;ENDFOLD
;FOLD LIN P197 CONT Vel=0.055 m/s CPDATP197 Tool[2] Base[8] ;%{PE}
;FOLD Parameters ;%{h}
;Params IlfProvider=kukaroboter.basistech.inlineforms.movement.old; Kuka.IsGlobalPoint=False; Kuka.PointName=P197; Kuka.BlendingEnabled=TRUE; Kuka.MoveDataName=CPDATP197; Kuka.VelocityPath=0.055; Kuka.CurrentCDSetIndex=0; Kuka.MovementParameterFieldEnabled=True; IlfCommand=LIN
;ENDFOLD
$BWDSTART = FALSE
LDAT_ACT=LCPDATP197
FDAT_ACT=FP197
BAS (#CP_PARAMS,0.055)
SET_CD_PARAMS (0)
LIN XP197 C_DIS

;ENDFOLD
;FOLD LIN P198 CONT Vel=0.12 m/s CPDATP198 Tool[2] Base[8] ;%{PE}
;FOLD Parameters ;%{h}
;Params IlfProvider=kukaroboter.basistech.inlineforms.movement.old; Kuka.IsGlobalPoint=False; Kuka.PointName=P198; Kuka.BlendingEnabled=TRUE; Kuka.MoveDataName=CPDATP198; Kuka.VelocityPath=0.12; Kuka.CurrentCDSetIndex=0; Kuka.MovementParameterFieldEnabled=True; IlfCommand=LIN
;ENDFOLD
$BWDSTART = FALSE
LDAT_ACT=LCPDATP198
FDAT_ACT=FP198
BAS (#CP_PARAMS,0.12)
SET_CD_PARAMS (0)
LIN XP198 C_DIS

;ENDFOLD
;FOLD LIN P199 CONT Vel=0.12 m/s CPDATP199 Tool[2] Base[8] ;%{PE}
;FOLD Parameters ;%{h}
;Params IlfProvider=kukaroboter.basistech.inlineforms.movement.old; Kuka.IsGlobalPoint=False; Kuka.PointName=P199; Kuka.BlendingEnabled=TRUE; Kuka.MoveDataName=CPDATP199; Kuka.VelocityPath=0.12; Kuka.CurrentCDSetIndex=0; Kuka.MovementParameterFieldEnabled=True; IlfCommand=LIN
;ENDFOLD
$BWDSTART = FALSE
LDAT_ACT=LCPDATP199
FDAT_ACT=FP199
BAS (#CP_PARAMS,0.12)
SET_CD_PARAMS (0)
LIN XP199 C_DIS

;ENDFOLD
;FOLD LIN P200 CONT Vel=0.12 m/s CPDATP200 Tool[2] Base[8] ;%{PE}
;FOLD Parameters ;%{h}
;Params IlfProvider=kukaroboter.basistech.inlineforms.movement.old; Kuka.IsGlobalPoint=False; Kuka.PointName=P200; Kuka.BlendingEnabled=TRUE; Kuka.MoveDataName=CPDATP200; Kuka.VelocityPath=0.12; Kuka.CurrentCDSetIndex=0; Kuka.MovementParameterFieldEnabled=True; IlfCommand=LIN
;ENDFOLD
$BWDSTART = FALSE
LDAT_ACT=LCPDATP200
FDAT_ACT=FP200
BAS (#CP_PARAMS,0.12)
SET_CD_PARAMS (0)
LIN XP200 C_DIS

;ENDFOLD
;FOLD LIN P201 CONT Vel=0.12 m/s CPDATP201 Tool[2] Base[8] ;%{PE}
;FOLD Parameters ;%{h}
;Params IlfProvider=kukaroboter.basistech.inlineforms.movement.old; Kuka.IsGlobalPoint=False; Kuka.PointName=P201; Kuka.BlendingEnabled=TRUE; Kuka.MoveDataName=CPDATP201; Kuka.VelocityPath=0.12; Kuka.CurrentCDSetIndex=0; Kuka.MovementParameterFieldEnabled=True; IlfCommand=LIN
;ENDFOLD
$BWDSTART = FALSE
LDAT_ACT=LCPDATP201
FDAT_ACT=FP201
BAS (#CP_PARAMS,0.12)
SET_CD_PARAMS (0)
LIN XP201 C_DIS

;ENDFOLD
;FOLD LIN P202 CONT Vel=0.081 m/s CPDATP202 Tool[2] Base[8] ;%{PE}
;FOLD Parameters ;%{h}
;Params IlfProvider=kukaroboter.basistech.inlineforms.movement.old; Kuka.IsGlobalPoint=False; Kuka.PointName=P202; Kuka.BlendingEnabled=TRUE; Kuka.MoveDataName=CPDATP202; Kuka.VelocityPath=0.081; Kuka.CurrentCDSetIndex=0; Kuka.MovementParameterFieldEnabled=True; IlfCommand=LIN
;ENDFOLD
$BWDSTART = FALSE
LDAT_ACT=LCPDATP202
FDAT_ACT=FP202
BAS (#CP_PARAMS,0.081)
SET_CD_PARAMS (0)
LIN XP202 C_DIS

;ENDFOLD
;FOLD LIN P203 CONT Vel=0.081 m/s CPDATP203 Tool[2] Base[8] ;%{PE}
;FOLD Parameters ;%{h}
;Params IlfProvider=kukaroboter.basistech.inlineforms.movement.old; Kuka.IsGlobalPoint=False; Kuka.PointName=P203; Kuka.BlendingEnabled=TRUE; Kuka.MoveDataName=CPDATP203; Kuka.VelocityPath=0.081; Kuka.CurrentCDSetIndex=0; Kuka.MovementParameterFieldEnabled=True; IlfCommand=LIN
;ENDFOLD
$BWDSTART = FALSE
LDAT_ACT=LCPDATP203
FDAT_ACT=FP203
BAS (#CP_PARAMS,0.081)
SET_CD_PARAMS (0)
LIN XP203 C_DIS

;ENDFOLD
;FOLD LIN P204 CONT Vel=0.081 m/s CPDATP204 Tool[2] Base[8] ;%{PE}
;FOLD Parameters ;%{h}
;Params IlfProvider=kukaroboter.basistech.inlineforms.movement.old; Kuka.IsGlobalPoint=False; Kuka.PointName=P204; Kuka.BlendingEnabled=TRUE; Kuka.MoveDataName=CPDATP204; Kuka.VelocityPath=0.081; Kuka.CurrentCDSetIndex=0; Kuka.MovementParameterFieldEnabled=True; IlfCommand=LIN
;ENDFOLD
$BWDSTART = FALSE
LDAT_ACT=LCPDATP204
FDAT_ACT=FP204
BAS (#CP_PARAMS,0.081)
SET_CD_PARAMS (0)
LIN XP204 C_DIS

;ENDFOLD
;FOLD LIN P205 CONT Vel=0.081 m/s CPDATP205 Tool[2] Base[8] ;%{PE}
;FOLD Parameters ;%{h}
;Params IlfProvider=kukaroboter.basistech.inlineforms.movement.old; Kuka.IsGlobalPoint=False; Kuka.PointName=P205; Kuka.BlendingEnabled=TRUE; Kuka.MoveDataName=CPDATP205; Kuka.VelocityPath=0.081; Kuka.CurrentCDSetIndex=0; Kuka.MovementParameterFieldEnabled=True; IlfCommand=LIN
;ENDFOLD
$BWDSTART = FALSE
LDAT_ACT=LCPDATP205
FDAT_ACT=FP205
BAS (#CP_PARAMS,0.081)
SET_CD_PARAMS (0)
LIN XP205 C_DIS

;ENDFOLD
;FOLD LIN P206 CONT Vel=0.147 m/s CPDATP206 Tool[2] Base[8] ;%{PE}
;FOLD Parameters ;%{h}
;Params IlfProvider=kukaroboter.basistech.inlineforms.movement.old; Kuka.IsGlobalPoint=False; Kuka.PointName=P206; Kuka.BlendingEnabled=TRUE; Kuka.MoveDataName=CPDATP206; Kuka.VelocityPath=0.147; Kuka.CurrentCDSetIndex=0; Kuka.MovementParameterFieldEnabled=True; IlfCommand=LIN
;ENDFOLD
$BWDSTART = FALSE
LDAT_ACT=LCPDATP206
FDAT_ACT=FP206
BAS (#CP_PARAMS,0.147)
SET_CD_PARAMS (0)
LIN XP206 C_DIS

;ENDFOLD
;FOLD LIN P207 CONT Vel=0.147 m/s CPDATP207 Tool[2] Base[8] ;%{PE}
;FOLD Parameters ;%{h}
;Params IlfProvider=kukaroboter.basistech.inlineforms.movement.old; Kuka.IsGlobalPoint=False; Kuka.PointName=P207; Kuka.BlendingEnabled=TRUE; Kuka.MoveDataName=CPDATP207; Kuka.VelocityPath=0.147; Kuka.CurrentCDSetIndex=0; Kuka.MovementParameterFieldEnabled=True; IlfCommand=LIN
;ENDFOLD
$BWDSTART = FALSE
LDAT_ACT=LCPDATP207
FDAT_ACT=FP207
BAS (#CP_PARAMS,0.147)
SET_CD_PARAMS (0)
LIN XP207 C_DIS

;ENDFOLD
;FOLD LIN P208 CONT Vel=0.147 m/s CPDATP208 Tool[2] Base[8] ;%{PE}
;FOLD Parameters ;%{h}
;Params IlfProvider=kukaroboter.basistech.inlineforms.movement.old; Kuka.IsGlobalPoint=False; Kuka.PointName=P208; Kuka.BlendingEnabled=TRUE; Kuka.MoveDataName=CPDATP208; Kuka.VelocityPath=0.147; Kuka.CurrentCDSetIndex=0; Kuka.MovementParameterFieldEnabled=True; IlfCommand=LIN
;ENDFOLD
$BWDSTART = FALSE
LDAT_ACT=LCPDATP208
FDAT_ACT=FP208
BAS (#CP_PARAMS,0.147)
SET_CD_PARAMS (0)
LIN XP208 C_DIS

;ENDFOLD
;FOLD LIN P209 CONT Vel=0.147 m/s CPDATP209 Tool[2] Base[8] ;%{PE}
;FOLD Parameters ;%{h}
;Params IlfProvider=kukaroboter.basistech.inlineforms.movement.old; Kuka.IsGlobalPoint=False; Kuka.PointName=P209; Kuka.BlendingEnabled=TRUE; Kuka.MoveDataName=CPDATP209; Kuka.VelocityPath=0.147; Kuka.CurrentCDSetIndex=0; Kuka.MovementParameterFieldEnabled=True; IlfCommand=LIN
;ENDFOLD
$BWDSTART = FALSE
LDAT_ACT=LCPDATP209
FDAT_ACT=FP209
BAS (#CP_PARAMS,0.147)
SET_CD_PARAMS (0)
LIN XP209 C_DIS

;ENDFOLD
;FOLD LIN P210 CONT Vel=0.076 m/s CPDATP210 Tool[2] Base[8] ;%{PE}
;FOLD Parameters ;%{h}
;Params IlfProvider=kukaroboter.basistech.inlineforms.movement.old; Kuka.IsGlobalPoint=False; Kuka.PointName=P210; Kuka.BlendingEnabled=TRUE; Kuka.MoveDataName=CPDATP210; Kuka.VelocityPath=0.076; Kuka.CurrentCDSetIndex=0; Kuka.MovementParameterFieldEnabled=True; IlfCommand=LIN
;ENDFOLD
$BWDSTART = FALSE
LDAT_ACT=LCPDATP210
FDAT_ACT=FP210
BAS (#CP_PARAMS,0.076)
SET_CD_PARAMS (0)
LIN XP210 C_DIS

;ENDFOLD
;FOLD LIN P211 CONT Vel=0.076 m/s CPDATP211 Tool[2] Base[8] ;%{PE}
;FOLD Parameters ;%{h}
;Params IlfProvider=kukaroboter.basistech.inlineforms.movement.old; Kuka.IsGlobalPoint=False; Kuka.PointName=P211; Kuka.BlendingEnabled=TRUE; Kuka.MoveDataName=CPDATP211; Kuka.VelocityPath=0.076; Kuka.CurrentCDSetIndex=0; Kuka.MovementParameterFieldEnabled=True; IlfCommand=LIN
;ENDFOLD
$BWDSTART = FALSE
LDAT_ACT=LCPDATP211
FDAT_ACT=FP211
BAS (#CP_PARAMS,0.076)
SET_CD_PARAMS (0)
LIN XP211 C_DIS

;ENDFOLD
;FOLD LIN P212 CONT Vel=0.076 m/s CPDATP212 Tool[2] Base[8] ;%{PE}
;FOLD Parameters ;%{h}
;Params IlfProvider=kukaroboter.basistech.inlineforms.movement.old; Kuka.IsGlobalPoint=False; Kuka.PointName=P212; Kuka.BlendingEnabled=TRUE; Kuka.MoveDataName=CPDATP212; Kuka.VelocityPath=0.076; Kuka.CurrentCDSetIndex=0; Kuka.MovementParameterFieldEnabled=True; IlfCommand=LIN
;ENDFOLD
$BWDSTART = FALSE
LDAT_ACT=LCPDATP212
FDAT_ACT=FP212
BAS (#CP_PARAMS,0.076)
SET_CD_PARAMS (0)
LIN XP212 C_DIS

;ENDFOLD
;FOLD LIN P213 CONT Vel=0.076 m/s CPDATP213 Tool[2] Base[8] ;%{PE}
;FOLD Parameters ;%{h}
;Params IlfProvider=kukaroboter.basistech.inlineforms.movement.old; Kuka.IsGlobalPoint=False; Kuka.PointName=P213; Kuka.BlendingEnabled=TRUE; Kuka.MoveDataName=CPDATP213; Kuka.VelocityPath=0.076; Kuka.CurrentCDSetIndex=0; Kuka.MovementParameterFieldEnabled=True; IlfCommand=LIN
;ENDFOLD
$BWDSTART = FALSE
LDAT_ACT=LCPDATP213
FDAT_ACT=FP213
BAS (#CP_PARAMS,0.076)
SET_CD_PARAMS (0)
LIN XP213 C_DIS

;ENDFOLD
;FOLD LIN P214 CONT Vel=0.126 m/s CPDATP214 Tool[2] Base[8] ;%{PE}
;FOLD Parameters ;%{h}
;Params IlfProvider=kukaroboter.basistech.inlineforms.movement.old; Kuka.IsGlobalPoint=False; Kuka.PointName=P214; Kuka.BlendingEnabled=TRUE; Kuka.MoveDataName=CPDATP214; Kuka.VelocityPath=0.126; Kuka.CurrentCDSetIndex=0; Kuka.MovementParameterFieldEnabled=True; IlfCommand=LIN
;ENDFOLD
$BWDSTART = FALSE
LDAT_ACT=LCPDATP214
FDAT_ACT=FP214
BAS (#CP_PARAMS,0.126)
SET_CD_PARAMS (0)
LIN XP214 C_DIS

;ENDFOLD
;FOLD LIN P215 CONT Vel=0.126 m/s CPDATP215 Tool[2] Base[8] ;%{PE}
;FOLD Parameters ;%{h}
;Params IlfProvider=kukaroboter.basistech.inlineforms.movement.old; Kuka.IsGlobalPoint=False; Kuka.PointName=P215; Kuka.BlendingEnabled=TRUE; Kuka.MoveDataName=CPDATP215; Kuka.VelocityPath=0.126; Kuka.CurrentCDSetIndex=0; Kuka.MovementParameterFieldEnabled=True; IlfCommand=LIN
;ENDFOLD
$BWDSTART = FALSE
LDAT_ACT=LCPDATP215
FDAT_ACT=FP215
BAS (#CP_PARAMS,0.126)
SET_CD_PARAMS (0)
LIN XP215 C_DIS

;ENDFOLD
;FOLD LIN P216 CONT Vel=0.126 m/s CPDATP216 Tool[2] Base[8] ;%{PE}
;FOLD Parameters ;%{h}
;Params IlfProvider=kukaroboter.basistech.inlineforms.movement.old; Kuka.IsGlobalPoint=False; Kuka.PointName=P216; Kuka.BlendingEnabled=TRUE; Kuka.MoveDataName=CPDATP216; Kuka.VelocityPath=0.126; Kuka.CurrentCDSetIndex=0; Kuka.MovementParameterFieldEnabled=True; IlfCommand=LIN
;ENDFOLD
$BWDSTART = FALSE
LDAT_ACT=LCPDATP216
FDAT_ACT=FP216
BAS (#CP_PARAMS,0.126)
SET_CD_PARAMS (0)
LIN XP216 C_DIS

;ENDFOLD
;FOLD LIN P217 CONT Vel=0.126 m/s CPDATP217 Tool[2] Base[8] ;%{PE}
;FOLD Parameters ;%{h}
;Params IlfProvider=kukaroboter.basistech.inlineforms.movement.old; Kuka.IsGlobalPoint=False; Kuka.PointName=P217; Kuka.BlendingEnabled=TRUE; Kuka.MoveDataName=CPDATP217; Kuka.VelocityPath=0.126; Kuka.CurrentCDSetIndex=0; Kuka.MovementParameterFieldEnabled=True; IlfCommand=LIN
;ENDFOLD
$BWDSTART = FALSE
LDAT_ACT=LCPDATP217
FDAT_ACT=FP217
BAS (#CP_PARAMS,0.126)
SET_CD_PARAMS (0)
LIN XP217 C_DIS

;ENDFOLD
;FOLD LIN P218 CONT Vel=0.13 m/s CPDATP218 Tool[2] Base[8] ;%{PE}
;FOLD Parameters ;%{h}
;Params IlfProvider=kukaroboter.basistech.inlineforms.movement.old; Kuka.IsGlobalPoint=False; Kuka.PointName=P218; Kuka.BlendingEnabled=TRUE; Kuka.MoveDataName=CPDATP218; Kuka.VelocityPath=0.13; Kuka.CurrentCDSetIndex=0; Kuka.MovementParameterFieldEnabled=True; IlfCommand=LIN
;ENDFOLD
$BWDSTART = FALSE
LDAT_ACT=LCPDATP218
FDAT_ACT=FP218
BAS (#CP_PARAMS,0.13)
SET_CD_PARAMS (0)
LIN XP218 C_DIS

;ENDFOLD
;FOLD LIN P219 CONT Vel=0.13 m/s CPDATP219 Tool[2] Base[8] ;%{PE}
;FOLD Parameters ;%{h}
;Params IlfProvider=kukaroboter.basistech.inlineforms.movement.old; Kuka.IsGlobalPoint=False; Kuka.PointName=P219; Kuka.BlendingEnabled=TRUE; Kuka.MoveDataName=CPDATP219; Kuka.VelocityPath=0.13; Kuka.CurrentCDSetIndex=0; Kuka.MovementParameterFieldEnabled=True; IlfCommand=LIN
;ENDFOLD
$BWDSTART = FALSE
LDAT_ACT=LCPDATP219
FDAT_ACT=FP219
BAS (#CP_PARAMS,0.13)
SET_CD_PARAMS (0)
LIN XP219 C_DIS

;ENDFOLD
;FOLD LIN P220 CONT Vel=0.13 m/s CPDATP220 Tool[2] Base[8] ;%{PE}
;FOLD Parameters ;%{h}
;Params IlfProvider=kukaroboter.basistech.inlineforms.movement.old; Kuka.IsGlobalPoint=False; Kuka.PointName=P220; Kuka.BlendingEnabled=TRUE; Kuka.MoveDataName=CPDATP220; Kuka.VelocityPath=0.13; Kuka.CurrentCDSetIndex=0; Kuka.MovementParameterFieldEnabled=True; IlfCommand=LIN
;ENDFOLD
$BWDSTART = FALSE
LDAT_ACT=LCPDATP220
FDAT_ACT=FP220
BAS (#CP_PARAMS,0.13)
SET_CD_PARAMS (0)
LIN XP220 C_DIS

;ENDFOLD
;FOLD LIN P221 CONT Vel=0.13 m/s CPDATP221 Tool[2] Base[8] ;%{PE}
;FOLD Parameters ;%{h}
;Params IlfProvider=kukaroboter.basistech.inlineforms.movement.old; Kuka.IsGlobalPoint=False; Kuka.PointName=P221; Kuka.BlendingEnabled=TRUE; Kuka.MoveDataName=CPDATP221; Kuka.VelocityPath=0.13; Kuka.CurrentCDSetIndex=0; Kuka.MovementParameterFieldEnabled=True; IlfCommand=LIN
;ENDFOLD
$BWDSTART = FALSE
LDAT_ACT=LCPDATP221
FDAT_ACT=FP221
BAS (#CP_PARAMS,0.13)
SET_CD_PARAMS (0)
LIN XP221 C_DIS

;ENDFOLD
;FOLD LIN P222 CONT Vel=0.106 m/s CPDATP222 Tool[2] Base[8] ;%{PE}
;FOLD Parameters ;%{h}
;Params IlfProvider=kukaroboter.basistech.inlineforms.movement.old; Kuka.IsGlobalPoint=False; Kuka.PointName=P222; Kuka.BlendingEnabled=TRUE; Kuka.MoveDataName=CPDATP222; Kuka.VelocityPath=0.106; Kuka.CurrentCDSetIndex=0; Kuka.MovementParameterFieldEnabled=True; IlfCommand=LIN
;ENDFOLD
$BWDSTART = FALSE
LDAT_ACT=LCPDATP222
FDAT_ACT=FP222
BAS (#CP_PARAMS,0.106)
SET_CD_PARAMS (0)
LIN XP222 C_DIS

;ENDFOLD
;FOLD LIN P223 CONT Vel=0.106 m/s CPDATP223 Tool[2] Base[8] ;%{PE}
;FOLD Parameters ;%{h}
;Params IlfProvider=kukaroboter.basistech.inlineforms.movement.old; Kuka.IsGlobalPoint=False; Kuka.PointName=P223; Kuka.BlendingEnabled=TRUE; Kuka.MoveDataName=CPDATP223; Kuka.VelocityPath=0.106; Kuka.CurrentCDSetIndex=0; Kuka.MovementParameterFieldEnabled=True; IlfCommand=LIN
;ENDFOLD
$BWDSTART = FALSE
LDAT_ACT=LCPDATP223
FDAT_ACT=FP223
BAS (#CP_PARAMS,0.106)
SET_CD_PARAMS (0)
LIN XP223 C_DIS

;ENDFOLD
;FOLD LIN P224 CONT Vel=0.106 m/s CPDATP224 Tool[2] Base[8] ;%{PE}
;FOLD Parameters ;%{h}
;Params IlfProvider=kukaroboter.basistech.inlineforms.movement.old; Kuka.IsGlobalPoint=False; Kuka.PointName=P224; Kuka.BlendingEnabled=TRUE; Kuka.MoveDataName=CPDATP224; Kuka.VelocityPath=0.106; Kuka.CurrentCDSetIndex=0; Kuka.MovementParameterFieldEnabled=True; IlfCommand=LIN
;ENDFOLD
$BWDSTART = FALSE
LDAT_ACT=LCPDATP224
FDAT_ACT=FP224
BAS (#CP_PARAMS,0.106)
SET_CD_PARAMS (0)
LIN XP224 C_DIS

;ENDFOLD
;FOLD LIN P225 CONT Vel=0.106 m/s CPDATP225 Tool[2] Base[8] ;%{PE}
;FOLD Parameters ;%{h}
;Params IlfProvider=kukaroboter.basistech.inlineforms.movement.old; Kuka.IsGlobalPoint=False; Kuka.PointName=P225; Kuka.BlendingEnabled=TRUE; Kuka.MoveDataName=CPDATP225; Kuka.VelocityPath=0.106; Kuka.CurrentCDSetIndex=0; Kuka.MovementParameterFieldEnabled=True; IlfCommand=LIN
;ENDFOLD
$BWDSTART = FALSE
LDAT_ACT=LCPDATP225
FDAT_ACT=FP225
BAS (#CP_PARAMS,0.106)
SET_CD_PARAMS (0)
LIN XP225 C_DIS

;ENDFOLD
;FOLD LIN P226 CONT Vel=0.145 m/s CPDATP226 Tool[2] Base[8] ;%{PE}
;FOLD Parameters ;%{h}
;Params IlfProvider=kukaroboter.basistech.inlineforms.movement.old; Kuka.IsGlobalPoint=False; Kuka.PointName=P226; Kuka.BlendingEnabled=TRUE; Kuka.MoveDataName=CPDATP226; Kuka.VelocityPath=0.145; Kuka.CurrentCDSetIndex=0; Kuka.MovementParameterFieldEnabled=True; IlfCommand=LIN
;ENDFOLD
$BWDSTART = FALSE
LDAT_ACT=LCPDATP226
FDAT_ACT=FP226
BAS (#CP_PARAMS,0.145)
SET_CD_PARAMS (0)
LIN XP226 C_DIS

;ENDFOLD
;FOLD LIN P227 CONT Vel=0.145 m/s CPDATP227 Tool[2] Base[8] ;%{PE}
;FOLD Parameters ;%{h}
;Params IlfProvider=kukaroboter.basistech.inlineforms.movement.old; Kuka.IsGlobalPoint=False; Kuka.PointName=P227; Kuka.BlendingEnabled=TRUE; Kuka.MoveDataName=CPDATP227; Kuka.VelocityPath=0.145; Kuka.CurrentCDSetIndex=0; Kuka.MovementParameterFieldEnabled=True; IlfCommand=LIN
;ENDFOLD
$BWDSTART = FALSE
LDAT_ACT=LCPDATP227
FDAT_ACT=FP227
BAS (#CP_PARAMS,0.145)
SET_CD_PARAMS (0)
LIN XP227 C_DIS

;ENDFOLD
;FOLD LIN P228 CONT Vel=0.145 m/s CPDATP228 Tool[2] Base[8] ;%{PE}
;FOLD Parameters ;%{h}
;Params IlfProvider=kukaroboter.basistech.inlineforms.movement.old; Kuka.IsGlobalPoint=False; Kuka.PointName=P228; Kuka.BlendingEnabled=TRUE; Kuka.MoveDataName=CPDATP228; Kuka.VelocityPath=0.145; Kuka.CurrentCDSetIndex=0; Kuka.MovementParameterFieldEnabled=True; IlfCommand=LIN
;ENDFOLD
$BWDSTART = FALSE
LDAT_ACT=LCPDATP228
FDAT_ACT=FP228
BAS (#CP_PARAMS,0.145)
SET_CD_PARAMS (0)
LIN XP228 C_DIS

;ENDFOLD
;FOLD LIN P229 CONT Vel=0.145 m/s CPDATP229 Tool[2] Base[8] ;%{PE}
;FOLD Parameters ;%{h}
;Params IlfProvider=kukaroboter.basistech.inlineforms.movement.old; Kuka.IsGlobalPoint=False; Kuka.PointName=P229; Kuka.BlendingEnabled=TRUE; Kuka.MoveDataName=CPDATP229; Kuka.VelocityPath=0.145; Kuka.CurrentCDSetIndex=0; Kuka.MovementParameterFieldEnabled=True; IlfCommand=LIN
;ENDFOLD
$BWDSTART = FALSE
LDAT_ACT=LCPDATP229
FDAT_ACT=FP229
BAS (#CP_PARAMS,0.145)
SET_CD_PARAMS (0)
LIN XP229 C_DIS

;ENDFOLD
;FOLD LIN P230 CONT Vel=0.1 m/s CPDATP230 Tool[2] Base[8] ;%{PE}
;FOLD Parameters ;%{h}
;Params IlfProvider=kukaroboter.basistech.inlineforms.movement.old; Kuka.IsGlobalPoint=False; Kuka.PointName=P230; Kuka.BlendingEnabled=TRUE; Kuka.MoveDataName=CPDATP230; Kuka.VelocityPath=0.1; Kuka.CurrentCDSetIndex=0; Kuka.MovementParameterFieldEnabled=True; IlfCommand=LIN
;ENDFOLD
$BWDSTART = FALSE
LDAT_ACT=LCPDATP230
FDAT_ACT=FP230
BAS (#CP_PARAMS,0.1)
SET_CD_PARAMS (0)
LIN XP230 C_DIS

;ENDFOLD
;FOLD LIN P231 CONT Vel=0.1 m/s CPDATP231 Tool[2] Base[8] ;%{PE}
;FOLD Parameters ;%{h}
;Params IlfProvider=kukaroboter.basistech.inlineforms.movement.old; Kuka.IsGlobalPoint=False; Kuka.PointName=P231; Kuka.BlendingEnabled=TRUE; Kuka.MoveDataName=CPDATP231; Kuka.VelocityPath=0.1; Kuka.CurrentCDSetIndex=0; Kuka.MovementParameterFieldEnabled=True; IlfCommand=LIN
;ENDFOLD
$BWDSTART = FALSE
LDAT_ACT=LCPDATP231
FDAT_ACT=FP231
BAS (#CP_PARAMS,0.1)
SET_CD_PARAMS (0)
LIN XP231 C_DIS

;ENDFOLD
;FOLD LIN P232 CONT Vel=0.1 m/s CPDATP232 Tool[2] Base[8] ;%{PE}
;FOLD Parameters ;%{h}
;Params IlfProvider=kukaroboter.basistech.inlineforms.movement.old; Kuka.IsGlobalPoint=False; Kuka.PointName=P232; Kuka.BlendingEnabled=TRUE; Kuka.MoveDataName=CPDATP232; Kuka.VelocityPath=0.1; Kuka.CurrentCDSetIndex=0; Kuka.MovementParameterFieldEnabled=True; IlfCommand=LIN
;ENDFOLD
$BWDSTART = FALSE
LDAT_ACT=LCPDATP232
FDAT_ACT=FP232
BAS (#CP_PARAMS,0.1)
SET_CD_PARAMS (0)
LIN XP232 C_DIS

;ENDFOLD
;FOLD LIN P233 CONT Vel=0.1 m/s CPDATP233 Tool[2] Base[8] ;%{PE}
;FOLD Parameters ;%{h}
;Params IlfProvider=kukaroboter.basistech.inlineforms.movement.old; Kuka.IsGlobalPoint=False; Kuka.PointName=P233; Kuka.BlendingEnabled=TRUE; Kuka.MoveDataName=CPDATP233; Kuka.VelocityPath=0.1; Kuka.CurrentCDSetIndex=0; Kuka.MovementParameterFieldEnabled=True; IlfCommand=LIN
;ENDFOLD
$BWDSTART = FALSE
LDAT_ACT=LCPDATP233
FDAT_ACT=FP233
BAS (#CP_PARAMS,0.1)
SET_CD_PARAMS (0)
LIN XP233 C_DIS

;ENDFOLD
;FOLD LIN P234 CONT Vel=0.13 m/s CPDATP234 Tool[2] Base[8] ;%{PE}
;FOLD Parameters ;%{h}
;Params IlfProvider=kukaroboter.basistech.inlineforms.movement.old; Kuka.IsGlobalPoint=False; Kuka.PointName=P234; Kuka.BlendingEnabled=TRUE; Kuka.MoveDataName=CPDATP234; Kuka.VelocityPath=0.13; Kuka.CurrentCDSetIndex=0; Kuka.MovementParameterFieldEnabled=True; IlfCommand=LIN
;ENDFOLD
$BWDSTART = FALSE
LDAT_ACT=LCPDATP234
FDAT_ACT=FP234
BAS (#CP_PARAMS,0.13)
SET_CD_PARAMS (0)
LIN XP234 C_DIS

;ENDFOLD
;FOLD LIN P235 CONT Vel=0.13 m/s CPDATP235 Tool[2] Base[8] ;%{PE}
;FOLD Parameters ;%{h}
;Params IlfProvider=kukaroboter.basistech.inlineforms.movement.old; Kuka.IsGlobalPoint=False; Kuka.PointName=P235; Kuka.BlendingEnabled=TRUE; Kuka.MoveDataName=CPDATP235; Kuka.VelocityPath=0.13; Kuka.CurrentCDSetIndex=0; Kuka.MovementParameterFieldEnabled=True; IlfCommand=LIN
;ENDFOLD
$BWDSTART = FALSE
LDAT_ACT=LCPDATP235
FDAT_ACT=FP235
BAS (#CP_PARAMS,0.13)
SET_CD_PARAMS (0)
LIN XP235 C_DIS

;ENDFOLD
;FOLD LIN P236 CONT Vel=0.13 m/s CPDATP236 Tool[2] Base[8] ;%{PE}
;FOLD Parameters ;%{h}
;Params IlfProvider=kukaroboter.basistech.inlineforms.movement.old; Kuka.IsGlobalPoint=False; Kuka.PointName=P236; Kuka.BlendingEnabled=TRUE; Kuka.MoveDataName=CPDATP236; Kuka.VelocityPath=0.13; Kuka.CurrentCDSetIndex=0; Kuka.MovementParameterFieldEnabled=True; IlfCommand=LIN
;ENDFOLD
$BWDSTART = FALSE
LDAT_ACT=LCPDATP236
FDAT_ACT=FP236
BAS (#CP_PARAMS,0.13)
SET_CD_PARAMS (0)
LIN XP236 C_DIS

;ENDFOLD
;FOLD LIN P237 CONT Vel=0.13 m/s CPDATP237 Tool[2] Base[8] ;%{PE}
;FOLD Parameters ;%{h}
;Params IlfProvider=kukaroboter.basistech.inlineforms.movement.old; Kuka.IsGlobalPoint=False; Kuka.PointName=P237; Kuka.BlendingEnabled=TRUE; Kuka.MoveDataName=CPDATP237; Kuka.VelocityPath=0.13; Kuka.CurrentCDSetIndex=0; Kuka.MovementParameterFieldEnabled=True; IlfCommand=LIN
;ENDFOLD
$BWDSTART = FALSE
LDAT_ACT=LCPDATP237
FDAT_ACT=FP237
BAS (#CP_PARAMS,0.13)
SET_CD_PARAMS (0)
LIN XP237 C_DIS

;ENDFOLD
;FOLD LIN P238 CONT Vel=0.091 m/s CPDATP238 Tool[2] Base[8] ;%{PE}
;FOLD Parameters ;%{h}
;Params IlfProvider=kukaroboter.basistech.inlineforms.movement.old; Kuka.IsGlobalPoint=False; Kuka.PointName=P238; Kuka.BlendingEnabled=TRUE; Kuka.MoveDataName=CPDATP238; Kuka.VelocityPath=0.091; Kuka.CurrentCDSetIndex=0; Kuka.MovementParameterFieldEnabled=True; IlfCommand=LIN
;ENDFOLD
$BWDSTART = FALSE
LDAT_ACT=LCPDATP238
FDAT_ACT=FP238
BAS (#CP_PARAMS,0.091)
SET_CD_PARAMS (0)
LIN XP238 C_DIS

;ENDFOLD
;FOLD LIN P239 CONT Vel=0.091 m/s CPDATP239 Tool[2] Base[8] ;%{PE}
;FOLD Parameters ;%{h}
;Params IlfProvider=kukaroboter.basistech.inlineforms.movement.old; Kuka.IsGlobalPoint=False; Kuka.PointName=P239; Kuka.BlendingEnabled=TRUE; Kuka.MoveDataName=CPDATP239; Kuka.VelocityPath=0.091; Kuka.CurrentCDSetIndex=0; Kuka.MovementParameterFieldEnabled=True; IlfCommand=LIN
;ENDFOLD
$BWDSTART = FALSE
LDAT_ACT=LCPDATP239
FDAT_ACT=FP239
BAS (#CP_PARAMS,0.091)
SET_CD_PARAMS (0)
LIN XP239 C_DIS

;ENDFOLD
;FOLD LIN P240 CONT Vel=0.091 m/s CPDATP240 Tool[2] Base[8] ;%{PE}
;FOLD Parameters ;%{h}
;Params IlfProvider=kukaroboter.basistech.inlineforms.movement.old; Kuka.IsGlobalPoint=False; Kuka.PointName=P240; Kuka.BlendingEnabled=TRUE; Kuka.MoveDataName=CPDATP240; Kuka.VelocityPath=0.091; Kuka.CurrentCDSetIndex=0; Kuka.MovementParameterFieldEnabled=True; IlfCommand=LIN
;ENDFOLD
$BWDSTART = FALSE
LDAT_ACT=LCPDATP240
FDAT_ACT=FP240
BAS (#CP_PARAMS,0.091)
SET_CD_PARAMS (0)
LIN XP240 C_DIS

;ENDFOLD
;FOLD LIN P241 CONT Vel=0.091 m/s CPDATP241 Tool[2] Base[8] ;%{PE}
;FOLD Parameters ;%{h}
;Params IlfProvider=kukaroboter.basistech.inlineforms.movement.old; Kuka.IsGlobalPoint=False; Kuka.PointName=P241; Kuka.BlendingEnabled=TRUE; Kuka.MoveDataName=CPDATP241; Kuka.VelocityPath=0.091; Kuka.CurrentCDSetIndex=0; Kuka.MovementParameterFieldEnabled=True; IlfCommand=LIN
;ENDFOLD
$BWDSTART = FALSE
LDAT_ACT=LCPDATP241
FDAT_ACT=FP241
BAS (#CP_PARAMS,0.091)
SET_CD_PARAMS (0)
LIN XP241 C_DIS

;ENDFOLD
;FOLD LIN P242 CONT Vel=0.5 m/s CPDATP242 Tool[2] Base[8] ;%{PE}
;FOLD Parameters ;%{h}
;Params IlfProvider=kukaroboter.basistech.inlineforms.movement.old; Kuka.IsGlobalPoint=False; Kuka.PointName=P242; Kuka.BlendingEnabled=TRUE; Kuka.MoveDataName=CPDATP242; Kuka.VelocityPath=0.5; Kuka.CurrentCDSetIndex=0; Kuka.MovementParameterFieldEnabled=True; IlfCommand=LIN
;ENDFOLD
$BWDSTART = FALSE
LDAT_ACT=LCPDATP242
FDAT_ACT=FP242
BAS (#CP_PARAMS,0.5)
SET_CD_PARAMS (0)
LIN XP242 C_DIS

;ENDFOLD
;FOLD LIN P243 CONT Vel=1.0 m/s CPDATP243 Tool[2] Base[8] ;%{PE}
;FOLD Parameters ;%{h}
;Params IlfProvider=kukaroboter.basistech.inlineforms.movement.old; Kuka.IsGlobalPoint=False; Kuka.PointName=P243; Kuka.BlendingEnabled=TRUE; Kuka.MoveDataName=CPDATP243; Kuka.VelocityPath=1.0; Kuka.CurrentCDSetIndex=0; Kuka.MovementParameterFieldEnabled=True; IlfCommand=LIN
;ENDFOLD
$BWDSTART = FALSE
LDAT_ACT=LCPDATP243
FDAT_ACT=FP243
BAS (#CP_PARAMS,1.0)
SET_CD_PARAMS (0)
LIN XP243 C_DIS

;ENDFOLD
;FOLD LIN P244 CONT Vel=1.0 m/s CPDATP244 Tool[2] Base[8] ;%{PE}
;FOLD Parameters ;%{h}
;Params IlfProvider=kukaroboter.basistech.inlineforms.movement.old; Kuka.IsGlobalPoint=False; Kuka.PointName=P244; Kuka.BlendingEnabled=TRUE; Kuka.MoveDataName=CPDATP244; Kuka.VelocityPath=1.0; Kuka.CurrentCDSetIndex=0; Kuka.MovementParameterFieldEnabled=True; IlfCommand=LIN
;ENDFOLD
$BWDSTART = FALSE
LDAT_ACT=LCPDATP244
FDAT_ACT=FP244
BAS (#CP_PARAMS,1.0)
SET_CD_PARAMS (0)
LIN XP244 C_DIS

;ENDFOLD
END
;End of routine {i}

; --- Routine for substrate 3 ---
DEF Routine_3()
;FOLD LIN P245 CONT Vel=1.0 m/s CPDATP245 Tool[2] Base[7] ;%{PE}
;FOLD Parameters ;%{h}
;Params IlfProvider=kukaroboter.basistech.inlineforms.movement.old; Kuka.IsGlobalPoint=False; Kuka.PointName=P245; Kuka.BlendingEnabled=TRUE; Kuka.MoveDataName=CPDATP245; Kuka.VelocityPath=1.0; Kuka.CurrentCDSetIndex=0; Kuka.MovementParameterFieldEnabled=True; IlfCommand=LIN
;ENDFOLD
$BWDSTART = FALSE
LDAT_ACT=LCPDATP245
FDAT_ACT=FP245
BAS (#CP_PARAMS,1.0)
SET_CD_PARAMS (0)
LIN XP245 C_DIS

;ENDFOLD
;FOLD LIN P246 CONT Vel=0.097 m/s CPDATP246 Tool[2] Base[7] ;%{PE}
;FOLD Parameters ;%{h}
;Params IlfProvider=kukaroboter.basistech.inlineforms.movement.old; Kuka.IsGlobalPoint=False; Kuka.PointName=P246; Kuka.BlendingEnabled=TRUE; Kuka.MoveDataName=CPDATP246; Kuka.VelocityPath=0.097; Kuka.CurrentCDSetIndex=0; Kuka.MovementParameterFieldEnabled=True; IlfCommand=LIN
;ENDFOLD
$BWDSTART = FALSE
LDAT_ACT=LCPDATP246
FDAT_ACT=FP246
BAS (#CP_PARAMS,0.097)
SET_CD_PARAMS (0)
LIN XP246 C_DIS

;ENDFOLD
;FOLD LIN P247 CONT Vel=0.097 m/s CPDATP247 Tool[2] Base[7] ;%{PE}
;FOLD Parameters ;%{h}
;Params IlfProvider=kukaroboter.basistech.inlineforms.movement.old; Kuka.IsGlobalPoint=False; Kuka.PointName=P247; Kuka.BlendingEnabled=TRUE; Kuka.MoveDataName=CPDATP247; Kuka.VelocityPath=0.097; Kuka.CurrentCDSetIndex=0; Kuka.MovementParameterFieldEnabled=True; IlfCommand=LIN
;ENDFOLD
$BWDSTART = FALSE
LDAT_ACT=LCPDATP247
FDAT_ACT=FP247
BAS (#CP_PARAMS,0.097)
SET_CD_PARAMS (0)
LIN XP247 C_DIS

;ENDFOLD
;FOLD LIN P248 CONT Vel=0.097 m/s CPDATP248 Tool[2] Base[7] ;%{PE}
;FOLD Parameters ;%{h}
;Params IlfProvider=kukaroboter.basistech.inlineforms.movement.old; Kuka.IsGlobalPoint=False; Kuka.PointName=P248; Kuka.BlendingEnabled=TRUE; Kuka.MoveDataName=CPDATP248; Kuka.VelocityPath=0.097; Kuka.CurrentCDSetIndex=0; Kuka.MovementParameterFieldEnabled=True; IlfCommand=LIN
;ENDFOLD
$BWDSTART = FALSE
LDAT_ACT=LCPDATP248
FDAT_ACT=FP248
BAS (#CP_PARAMS,0.097)
SET_CD_PARAMS (0)
LIN XP248 C_DIS

;ENDFOLD
;FOLD LIN P249 CONT Vel=0.097 m/s CPDATP249 Tool[2] Base[7] ;%{PE}
;FOLD Parameters ;%{h}
;Params IlfProvider=kukaroboter.basistech.inlineforms.movement.old; Kuka.IsGlobalPoint=False; Kuka.PointName=P249; Kuka.BlendingEnabled=TRUE; Kuka.MoveDataName=CPDATP249; Kuka.VelocityPath=0.097; Kuka.CurrentCDSetIndex=0; Kuka.MovementParameterFieldEnabled=True; IlfCommand=LIN
;ENDFOLD
$BWDSTART = FALSE
LDAT_ACT=LCPDATP249
FDAT_ACT=FP249
BAS (#CP_PARAMS,0.097)
SET_CD_PARAMS (0)
LIN XP249 C_DIS

;ENDFOLD
;FOLD LIN P250 CONT Vel=0.144 m/s CPDATP250 Tool[2] Base[7] ;%{PE}
;FOLD Parameters ;%{h}
;Params IlfProvider=kukaroboter.basistech.inlineforms.movement.old; Kuka.IsGlobalPoint=False; Kuka.PointName=P250; Kuka.BlendingEnabled=TRUE; Kuka.MoveDataName=CPDATP250; Kuka.VelocityPath=0.144; Kuka.CurrentCDSetIndex=0; Kuka.MovementParameterFieldEnabled=True; IlfCommand=LIN
;ENDFOLD
$BWDSTART = FALSE
LDAT_ACT=LCPDATP250
FDAT_ACT=FP250
BAS (#CP_PARAMS,0.144)
SET_CD_PARAMS (0)
LIN XP250 C_DIS

;ENDFOLD
;FOLD LIN P251 CONT Vel=0.144 m/s CPDATP251 Tool[2] Base[7] ;%{PE}
;FOLD Parameters ;%{h}
;Params IlfProvider=kukaroboter.basistech.inlineforms.movement.old; Kuka.IsGlobalPoint=False; Kuka.PointName=P251; Kuka.BlendingEnabled=TRUE; Kuka.MoveDataName=CPDATP251; Kuka.VelocityPath=0.144; Kuka.CurrentCDSetIndex=0; Kuka.MovementParameterFieldEnabled=True; IlfCommand=LIN
;ENDFOLD
$BWDSTART = FALSE
LDAT_ACT=LCPDATP251
FDAT_ACT=FP251
BAS (#CP_PARAMS,0.144)
SET_CD_PARAMS (0)
LIN XP251 C_DIS

;ENDFOLD
;FOLD LIN P252 CONT Vel=0.144 m/s CPDATP252 Tool[2] Base[7] ;%{PE}
;FOLD Parameters ;%{h}
;Params IlfProvider=kukaroboter.basistech.inlineforms.movement.old; Kuka.IsGlobalPoint=False; Kuka.PointName=P252; Kuka.BlendingEnabled=TRUE; Kuka.MoveDataName=CPDATP252; Kuka.VelocityPath=0.144; Kuka.CurrentCDSetIndex=0; Kuka.MovementParameterFieldEnabled=True; IlfCommand=LIN
;ENDFOLD
$BWDSTART = FALSE
LDAT_ACT=LCPDATP252
FDAT_ACT=FP252
BAS (#CP_PARAMS,0.144)
SET_CD_PARAMS (0)
LIN XP252 C_DIS

;ENDFOLD
;FOLD LIN P253 CONT Vel=0.144 m/s CPDATP253 Tool[2] Base[7] ;%{PE}
;FOLD Parameters ;%{h}
;Params IlfProvider=kukaroboter.basistech.inlineforms.movement.old; Kuka.IsGlobalPoint=False; Kuka.PointName=P253; Kuka.BlendingEnabled=TRUE; Kuka.MoveDataName=CPDATP253; Kuka.VelocityPath=0.144; Kuka.CurrentCDSetIndex=0; Kuka.MovementParameterFieldEnabled=True; IlfCommand=LIN
;ENDFOLD
$BWDSTART = FALSE
LDAT_ACT=LCPDATP253
FDAT_ACT=FP253
BAS (#CP_PARAMS,0.144)
SET_CD_PARAMS (0)
LIN XP253 C_DIS

;ENDFOLD
;FOLD LIN P254 CONT Vel=0.084 m/s CPDATP254 Tool[2] Base[7] ;%{PE}
;FOLD Parameters ;%{h}
;Params IlfProvider=kukaroboter.basistech.inlineforms.movement.old; Kuka.IsGlobalPoint=False; Kuka.PointName=P254; Kuka.BlendingEnabled=TRUE; Kuka.MoveDataName=CPDATP254; Kuka.VelocityPath=0.084; Kuka.CurrentCDSetIndex=0; Kuka.MovementParameterFieldEnabled=True; IlfCommand=LIN
;ENDFOLD
$BWDSTART = FALSE
LDAT_ACT=LCPDATP254
FDAT_ACT=FP254
BAS (#CP_PARAMS,0.084)
SET_CD_PARAMS (0)
LIN XP254 C_DIS

;ENDFOLD
;FOLD LIN P255 CONT Vel=0.084 m/s CPDATP255 Tool[2] Base[7] ;%{PE}
;FOLD Parameters ;%{h}
;Params IlfProvider=kukaroboter.basistech.inlineforms.movement.old; Kuka.IsGlobalPoint=False; Kuka.PointName=P255; Kuka.BlendingEnabled=TRUE; Kuka.MoveDataName=CPDATP255; Kuka.VelocityPath=0.084; Kuka.CurrentCDSetIndex=0; Kuka.MovementParameterFieldEnabled=True; IlfCommand=LIN
;ENDFOLD
$BWDSTART = FALSE
LDAT_ACT=LCPDATP255
FDAT_ACT=FP255
BAS (#CP_PARAMS,0.084)
SET_CD_PARAMS (0)
LIN XP255 C_DIS

;ENDFOLD
;FOLD LIN P256 CONT Vel=0.084 m/s CPDATP256 Tool[2] Base[7] ;%{PE}
;FOLD Parameters ;%{h}
;Params IlfProvider=kukaroboter.basistech.inlineforms.movement.old; Kuka.IsGlobalPoint=False; Kuka.PointName=P256; Kuka.BlendingEnabled=TRUE; Kuka.MoveDataName=CPDATP256; Kuka.VelocityPath=0.084; Kuka.CurrentCDSetIndex=0; Kuka.MovementParameterFieldEnabled=True; IlfCommand=LIN
;ENDFOLD
$BWDSTART = FALSE
LDAT_ACT=LCPDATP256
FDAT_ACT=FP256
BAS (#CP_PARAMS,0.084)
SET_CD_PARAMS (0)
LIN XP256 C_DIS

;ENDFOLD
;FOLD LIN P257 CONT Vel=0.084 m/s CPDATP257 Tool[2] Base[7] ;%{PE}
;FOLD Parameters ;%{h}
;Params IlfProvider=kukaroboter.basistech.inlineforms.movement.old; Kuka.IsGlobalPoint=False; Kuka.PointName=P257; Kuka.BlendingEnabled=TRUE; Kuka.MoveDataName=CPDATP257; Kuka.VelocityPath=0.084; Kuka.CurrentCDSetIndex=0; Kuka.MovementParameterFieldEnabled=True; IlfCommand=LIN
;ENDFOLD
$BWDSTART = FALSE
LDAT_ACT=LCPDATP257
FDAT_ACT=FP257
BAS (#CP_PARAMS,0.084)
SET_CD_PARAMS (0)
LIN XP257 C_DIS

;ENDFOLD
;FOLD LIN P258 CONT Vel=0.05 m/s CPDATP258 Tool[2] Base[7] ;%{PE}
;FOLD Parameters ;%{h}
;Params IlfProvider=kukaroboter.basistech.inlineforms.movement.old; Kuka.IsGlobalPoint=False; Kuka.PointName=P258; Kuka.BlendingEnabled=TRUE; Kuka.MoveDataName=CPDATP258; Kuka.VelocityPath=0.05; Kuka.CurrentCDSetIndex=0; Kuka.MovementParameterFieldEnabled=True; IlfCommand=LIN
;ENDFOLD
$BWDSTART = FALSE
LDAT_ACT=LCPDATP258
FDAT_ACT=FP258
BAS (#CP_PARAMS,0.05)
SET_CD_PARAMS (0)
LIN XP258 C_DIS

;ENDFOLD
;FOLD LIN P259 CONT Vel=0.05 m/s CPDATP259 Tool[2] Base[7] ;%{PE}
;FOLD Parameters ;%{h}
;Params IlfProvider=kukaroboter.basistech.inlineforms.movement.old; Kuka.IsGlobalPoint=False; Kuka.PointName=P259; Kuka.BlendingEnabled=TRUE; Kuka.MoveDataName=CPDATP259; Kuka.VelocityPath=0.05; Kuka.CurrentCDSetIndex=0; Kuka.MovementParameterFieldEnabled=True; IlfCommand=LIN
;ENDFOLD
$BWDSTART = FALSE
LDAT_ACT=LCPDATP259
FDAT_ACT=FP259
BAS (#CP_PARAMS,0.05)
SET_CD_PARAMS (0)
LIN XP259 C_DIS

;ENDFOLD
;FOLD LIN P260 CONT Vel=0.05 m/s CPDATP260 Tool[2] Base[7] ;%{PE}
;FOLD Parameters ;%{h}
;Params IlfProvider=kukaroboter.basistech.inlineforms.movement.old; Kuka.IsGlobalPoint=False; Kuka.PointName=P260; Kuka.BlendingEnabled=TRUE; Kuka.MoveDataName=CPDATP260; Kuka.VelocityPath=0.05; Kuka.CurrentCDSetIndex=0; Kuka.MovementParameterFieldEnabled=True; IlfCommand=LIN
;ENDFOLD
$BWDSTART = FALSE
LDAT_ACT=LCPDATP260
FDAT_ACT=FP260
BAS (#CP_PARAMS,0.05)
SET_CD_PARAMS (0)
LIN XP260 C_DIS

;ENDFOLD
;FOLD LIN P261 CONT Vel=0.05 m/s CPDATP261 Tool[2] Base[7] ;%{PE}
;FOLD Parameters ;%{h}
;Params IlfProvider=kukaroboter.basistech.inlineforms.movement.old; Kuka.IsGlobalPoint=False; Kuka.PointName=P261; Kuka.BlendingEnabled=TRUE; Kuka.MoveDataName=CPDATP261; Kuka.VelocityPath=0.05; Kuka.CurrentCDSetIndex=0; Kuka.MovementParameterFieldEnabled=True; IlfCommand=LIN
;ENDFOLD
$BWDSTART = FALSE
LDAT_ACT=LCPDATP261
FDAT_ACT=FP261
BAS (#CP_PARAMS,0.05)
SET_CD_PARAMS (0)
LIN XP261 C_DIS

;ENDFOLD
;FOLD LIN P262 CONT Vel=0.077 m/s CPDATP262 Tool[2] Base[7] ;%{PE}
;FOLD Parameters ;%{h}
;Params IlfProvider=kukaroboter.basistech.inlineforms.movement.old; Kuka.IsGlobalPoint=False; Kuka.PointName=P262; Kuka.BlendingEnabled=TRUE; Kuka.MoveDataName=CPDATP262; Kuka.VelocityPath=0.077; Kuka.CurrentCDSetIndex=0; Kuka.MovementParameterFieldEnabled=True; IlfCommand=LIN
;ENDFOLD
$BWDSTART = FALSE
LDAT_ACT=LCPDATP262
FDAT_ACT=FP262
BAS (#CP_PARAMS,0.077)
SET_CD_PARAMS (0)
LIN XP262 C_DIS

;ENDFOLD
;FOLD LIN P263 CONT Vel=0.077 m/s CPDATP263 Tool[2] Base[7] ;%{PE}
;FOLD Parameters ;%{h}
;Params IlfProvider=kukaroboter.basistech.inlineforms.movement.old; Kuka.IsGlobalPoint=False; Kuka.PointName=P263; Kuka.BlendingEnabled=TRUE; Kuka.MoveDataName=CPDATP263; Kuka.VelocityPath=0.077; Kuka.CurrentCDSetIndex=0; Kuka.MovementParameterFieldEnabled=True; IlfCommand=LIN
;ENDFOLD
$BWDSTART = FALSE
LDAT_ACT=LCPDATP263
FDAT_ACT=FP263
BAS (#CP_PARAMS,0.077)
SET_CD_PARAMS (0)
LIN XP263 C_DIS

;ENDFOLD
;FOLD LIN P264 CONT Vel=0.077 m/s CPDATP264 Tool[2] Base[7] ;%{PE}
;FOLD Parameters ;%{h}
;Params IlfProvider=kukaroboter.basistech.inlineforms.movement.old; Kuka.IsGlobalPoint=False; Kuka.PointName=P264; Kuka.BlendingEnabled=TRUE; Kuka.MoveDataName=CPDATP264; Kuka.VelocityPath=0.077; Kuka.CurrentCDSetIndex=0; Kuka.MovementParameterFieldEnabled=True; IlfCommand=LIN
;ENDFOLD
$BWDSTART = FALSE
LDAT_ACT=LCPDATP264
FDAT_ACT=FP264
BAS (#CP_PARAMS,0.077)
SET_CD_PARAMS (0)
LIN XP264 C_DIS

;ENDFOLD
;FOLD LIN P265 CONT Vel=0.077 m/s CPDATP265 Tool[2] Base[7] ;%{PE}
;FOLD Parameters ;%{h}
;Params IlfProvider=kukaroboter.basistech.inlineforms.movement.old; Kuka.IsGlobalPoint=False; Kuka.PointName=P265; Kuka.BlendingEnabled=TRUE; Kuka.MoveDataName=CPDATP265; Kuka.VelocityPath=0.077; Kuka.CurrentCDSetIndex=0; Kuka.MovementParameterFieldEnabled=True; IlfCommand=LIN
;ENDFOLD
$BWDSTART = FALSE
LDAT_ACT=LCPDATP265
FDAT_ACT=FP265
BAS (#CP_PARAMS,0.077)
SET_CD_PARAMS (0)
LIN XP265 C_DIS

;ENDFOLD
;FOLD LIN P266 CONT Vel=0.091 m/s CPDATP266 Tool[2] Base[7] ;%{PE}
;FOLD Parameters ;%{h}
;Params IlfProvider=kukaroboter.basistech.inlineforms.movement.old; Kuka.IsGlobalPoint=False; Kuka.PointName=P266; Kuka.BlendingEnabled=TRUE; Kuka.MoveDataName=CPDATP266; Kuka.VelocityPath=0.091; Kuka.CurrentCDSetIndex=0; Kuka.MovementParameterFieldEnabled=True; IlfCommand=LIN
;ENDFOLD
$BWDSTART = FALSE
LDAT_ACT=LCPDATP266
FDAT_ACT=FP266
BAS (#CP_PARAMS,0.091)
SET_CD_PARAMS (0)
LIN XP266 C_DIS

;ENDFOLD
;FOLD LIN P267 CONT Vel=0.091 m/s CPDATP267 Tool[2] Base[7] ;%{PE}
;FOLD Parameters ;%{h}
;Params IlfProvider=kukaroboter.basistech.inlineforms.movement.old; Kuka.IsGlobalPoint=False; Kuka.PointName=P267; Kuka.BlendingEnabled=TRUE; Kuka.MoveDataName=CPDATP267; Kuka.VelocityPath=0.091; Kuka.CurrentCDSetIndex=0; Kuka.MovementParameterFieldEnabled=True; IlfCommand=LIN
;ENDFOLD
$BWDSTART = FALSE
LDAT_ACT=LCPDATP267
FDAT_ACT=FP267
BAS (#CP_PARAMS,0.091)
SET_CD_PARAMS (0)
LIN XP267 C_DIS

;ENDFOLD
;FOLD LIN P268 CONT Vel=0.091 m/s CPDATP268 Tool[2] Base[7] ;%{PE}
;FOLD Parameters ;%{h}
;Params IlfProvider=kukaroboter.basistech.inlineforms.movement.old; Kuka.IsGlobalPoint=False; Kuka.PointName=P268; Kuka.BlendingEnabled=TRUE; Kuka.MoveDataName=CPDATP268; Kuka.VelocityPath=0.091; Kuka.CurrentCDSetIndex=0; Kuka.MovementParameterFieldEnabled=True; IlfCommand=LIN
;ENDFOLD
$BWDSTART = FALSE
LDAT_ACT=LCPDATP268
FDAT_ACT=FP268
BAS (#CP_PARAMS,0.091)
SET_CD_PARAMS (0)
LIN XP268 C_DIS

;ENDFOLD
;FOLD LIN P269 CONT Vel=0.091 m/s CPDATP269 Tool[2] Base[7] ;%{PE}
;FOLD Parameters ;%{h}
;Params IlfProvider=kukaroboter.basistech.inlineforms.movement.old; Kuka.IsGlobalPoint=False; Kuka.PointName=P269; Kuka.BlendingEnabled=TRUE; Kuka.MoveDataName=CPDATP269; Kuka.VelocityPath=0.091; Kuka.CurrentCDSetIndex=0; Kuka.MovementParameterFieldEnabled=True; IlfCommand=LIN
;ENDFOLD
$BWDSTART = FALSE
LDAT_ACT=LCPDATP269
FDAT_ACT=FP269
BAS (#CP_PARAMS,0.091)
SET_CD_PARAMS (0)
LIN XP269 C_DIS

;ENDFOLD
;FOLD LIN P270 CONT Vel=0.058 m/s CPDATP270 Tool[2] Base[7] ;%{PE}
;FOLD Parameters ;%{h}
;Params IlfProvider=kukaroboter.basistech.inlineforms.movement.old; Kuka.IsGlobalPoint=False; Kuka.PointName=P270; Kuka.BlendingEnabled=TRUE; Kuka.MoveDataName=CPDATP270; Kuka.VelocityPath=0.058; Kuka.CurrentCDSetIndex=0; Kuka.MovementParameterFieldEnabled=True; IlfCommand=LIN
;ENDFOLD
$BWDSTART = FALSE
LDAT_ACT=LCPDATP270
FDAT_ACT=FP270
BAS (#CP_PARAMS,0.058)
SET_CD_PARAMS (0)
LIN XP270 C_DIS

;ENDFOLD
;FOLD LIN P271 CONT Vel=0.058 m/s CPDATP271 Tool[2] Base[7] ;%{PE}
;FOLD Parameters ;%{h}
;Params IlfProvider=kukaroboter.basistech.inlineforms.movement.old; Kuka.IsGlobalPoint=False; Kuka.PointName=P271; Kuka.BlendingEnabled=TRUE; Kuka.MoveDataName=CPDATP271; Kuka.VelocityPath=0.058; Kuka.CurrentCDSetIndex=0; Kuka.MovementParameterFieldEnabled=True; IlfCommand=LIN
;ENDFOLD
$BWDSTART = FALSE
LDAT_ACT=LCPDATP271
FDAT_ACT=FP271
BAS (#CP_PARAMS,0.058)
SET_CD_PARAMS (0)
LIN XP271 C_DIS

;ENDFOLD
;FOLD LIN P272 CONT Vel=0.058 m/s CPDATP272 Tool[2] Base[7] ;%{PE}
;FOLD Parameters ;%{h}
;Params IlfProvider=kukaroboter.basistech.inlineforms.movement.old; Kuka.IsGlobalPoint=False; Kuka.PointName=P272; Kuka.BlendingEnabled=TRUE; Kuka.MoveDataName=CPDATP272; Kuka.VelocityPath=0.058; Kuka.CurrentCDSetIndex=0; Kuka.MovementParameterFieldEnabled=True; IlfCommand=LIN
;ENDFOLD
$BWDSTART = FALSE
LDAT_ACT=LCPDATP272
FDAT_ACT=FP272
BAS (#CP_PARAMS,0.058)
SET_CD_PARAMS (0)
LIN XP272 C_DIS

;ENDFOLD
;FOLD LIN P273 CONT Vel=0.058 m/s CPDATP273 Tool[2] Base[7] ;%{PE}
;FOLD Parameters ;%{h}
;Params IlfProvider=kukaroboter.basistech.inlineforms.movement.old; Kuka.IsGlobalPoint=False; Kuka.PointName=P273; Kuka.BlendingEnabled=TRUE; Kuka.MoveDataName=CPDATP273; Kuka.VelocityPath=0.058; Kuka.CurrentCDSetIndex=0; Kuka.MovementParameterFieldEnabled=True; IlfCommand=LIN
;ENDFOLD
$BWDSTART = FALSE
LDAT_ACT=LCPDATP273
FDAT_ACT=FP273
BAS (#CP_PARAMS,0.058)
SET_CD_PARAMS (0)
LIN XP273 C_DIS

;ENDFOLD
;FOLD LIN P274 CONT Vel=0.08 m/s CPDATP274 Tool[2] Base[7] ;%{PE}
;FOLD Parameters ;%{h}
;Params IlfProvider=kukaroboter.basistech.inlineforms.movement.old; Kuka.IsGlobalPoint=False; Kuka.PointName=P274; Kuka.BlendingEnabled=TRUE; Kuka.MoveDataName=CPDATP274; Kuka.VelocityPath=0.08; Kuka.CurrentCDSetIndex=0; Kuka.MovementParameterFieldEnabled=True; IlfCommand=LIN
;ENDFOLD
$BWDSTART = FALSE
LDAT_ACT=LCPDATP274
FDAT_ACT=FP274
BAS (#CP_PARAMS,0.08)
SET_CD_PARAMS (0)
LIN XP274 C_DIS

;ENDFOLD
;FOLD LIN P275 CONT Vel=0.08 m/s CPDATP275 Tool[2] Base[7] ;%{PE}
;FOLD Parameters ;%{h}
;Params IlfProvider=kukaroboter.basistech.inlineforms.movement.old; Kuka.IsGlobalPoint=False; Kuka.PointName=P275; Kuka.BlendingEnabled=TRUE; Kuka.MoveDataName=CPDATP275; Kuka.VelocityPath=0.08; Kuka.CurrentCDSetIndex=0; Kuka.MovementParameterFieldEnabled=True; IlfCommand=LIN
;ENDFOLD
$BWDSTART = FALSE
LDAT_ACT=LCPDATP275
FDAT_ACT=FP275
BAS (#CP_PARAMS,0.08)
SET_CD_PARAMS (0)
LIN XP275 C_DIS

;ENDFOLD
;FOLD LIN P276 CONT Vel=0.08 m/s CPDATP276 Tool[2] Base[7] ;%{PE}
;FOLD Parameters ;%{h}
;Params IlfProvider=kukaroboter.basistech.inlineforms.movement.old; Kuka.IsGlobalPoint=False; Kuka.PointName=P276; Kuka.BlendingEnabled=TRUE; Kuka.MoveDataName=CPDATP276; Kuka.VelocityPath=0.08; Kuka.CurrentCDSetIndex=0; Kuka.MovementParameterFieldEnabled=True; IlfCommand=LIN
;ENDFOLD
$BWDSTART = FALSE
LDAT_ACT=LCPDATP276
FDAT_ACT=FP276
BAS (#CP_PARAMS,0.08)
SET_CD_PARAMS (0)
LIN XP276 C_DIS

;ENDFOLD
;FOLD LIN P277 CONT Vel=0.08 m/s CPDATP277 Tool[2] Base[7] ;%{PE}
;FOLD Parameters ;%{h}
;Params IlfProvider=kukaroboter.basistech.inlineforms.movement.old; Kuka.IsGlobalPoint=False; Kuka.PointName=P277; Kuka.BlendingEnabled=TRUE; Kuka.MoveDataName=CPDATP277; Kuka.VelocityPath=0.08; Kuka.CurrentCDSetIndex=0; Kuka.MovementParameterFieldEnabled=True; IlfCommand=LIN
;ENDFOLD
$BWDSTART = FALSE
LDAT_ACT=LCPDATP277
FDAT_ACT=FP277
BAS (#CP_PARAMS,0.08)
SET_CD_PARAMS (0)
LIN XP277 C_DIS

;ENDFOLD
;FOLD LIN P278 CONT Vel=0.079 m/s CPDATP278 Tool[2] Base[7] ;%{PE}
;FOLD Parameters ;%{h}
;Params IlfProvider=kukaroboter.basistech.inlineforms.movement.old; Kuka.IsGlobalPoint=False; Kuka.PointName=P278; Kuka.BlendingEnabled=TRUE; Kuka.MoveDataName=CPDATP278; Kuka.VelocityPath=0.079; Kuka.CurrentCDSetIndex=0; Kuka.MovementParameterFieldEnabled=True; IlfCommand=LIN
;ENDFOLD
$BWDSTART = FALSE
LDAT_ACT=LCPDATP278
FDAT_ACT=FP278
BAS (#CP_PARAMS,0.079)
SET_CD_PARAMS (0)
LIN XP278 C_DIS

;ENDFOLD
;FOLD LIN P279 CONT Vel=0.079 m/s CPDATP279 Tool[2] Base[7] ;%{PE}
;FOLD Parameters ;%{h}
;Params IlfProvider=kukaroboter.basistech.inlineforms.movement.old; Kuka.IsGlobalPoint=False; Kuka.PointName=P279; Kuka.BlendingEnabled=TRUE; Kuka.MoveDataName=CPDATP279; Kuka.VelocityPath=0.079; Kuka.CurrentCDSetIndex=0; Kuka.MovementParameterFieldEnabled=True; IlfCommand=LIN
;ENDFOLD
$BWDSTART = FALSE
LDAT_ACT=LCPDATP279
FDAT_ACT=FP279
BAS (#CP_PARAMS,0.079)
SET_CD_PARAMS (0)
LIN XP279 C_DIS

;ENDFOLD
;FOLD LIN P280 CONT Vel=0.079 m/s CPDATP280 Tool[2] Base[7] ;%{PE}
;FOLD Parameters ;%{h}
;Params IlfProvider=kukaroboter.basistech.inlineforms.movement.old; Kuka.IsGlobalPoint=False; Kuka.PointName=P280; Kuka.BlendingEnabled=TRUE; Kuka.MoveDataName=CPDATP280; Kuka.VelocityPath=0.079; Kuka.CurrentCDSetIndex=0; Kuka.MovementParameterFieldEnabled=True; IlfCommand=LIN
;ENDFOLD
$BWDSTART = FALSE
LDAT_ACT=LCPDATP280
FDAT_ACT=FP280
BAS (#CP_PARAMS,0.079)
SET_CD_PARAMS (0)
LIN XP280 C_DIS

;ENDFOLD
;FOLD LIN P281 CONT Vel=0.079 m/s CPDATP281 Tool[2] Base[7] ;%{PE}
;FOLD Parameters ;%{h}
;Params IlfProvider=kukaroboter.basistech.inlineforms.movement.old; Kuka.IsGlobalPoint=False; Kuka.PointName=P281; Kuka.BlendingEnabled=TRUE; Kuka.MoveDataName=CPDATP281; Kuka.VelocityPath=0.079; Kuka.CurrentCDSetIndex=0; Kuka.MovementParameterFieldEnabled=True; IlfCommand=LIN
;ENDFOLD
$BWDSTART = FALSE
LDAT_ACT=LCPDATP281
FDAT_ACT=FP281
BAS (#CP_PARAMS,0.079)
SET_CD_PARAMS (0)
LIN XP281 C_DIS

;ENDFOLD
;FOLD LIN P282 CONT Vel=0.134 m/s CPDATP282 Tool[2] Base[7] ;%{PE}
;FOLD Parameters ;%{h}
;Params IlfProvider=kukaroboter.basistech.inlineforms.movement.old; Kuka.IsGlobalPoint=False; Kuka.PointName=P282; Kuka.BlendingEnabled=TRUE; Kuka.MoveDataName=CPDATP282; Kuka.VelocityPath=0.134; Kuka.CurrentCDSetIndex=0; Kuka.MovementParameterFieldEnabled=True; IlfCommand=LIN
;ENDFOLD
$BWDSTART = FALSE
LDAT_ACT=LCPDATP282
FDAT_ACT=FP282
BAS (#CP_PARAMS,0.134)
SET_CD_PARAMS (0)
LIN XP282 C_DIS

;ENDFOLD
;FOLD LIN P283 CONT Vel=0.134 m/s CPDATP283 Tool[2] Base[7] ;%{PE}
;FOLD Parameters ;%{h}
;Params IlfProvider=kukaroboter.basistech.inlineforms.movement.old; Kuka.IsGlobalPoint=False; Kuka.PointName=P283; Kuka.BlendingEnabled=TRUE; Kuka.MoveDataName=CPDATP283; Kuka.VelocityPath=0.134; Kuka.CurrentCDSetIndex=0; Kuka.MovementParameterFieldEnabled=True; IlfCommand=LIN
;ENDFOLD
$BWDSTART = FALSE
LDAT_ACT=LCPDATP283
FDAT_ACT=FP283
BAS (#CP_PARAMS,0.134)
SET_CD_PARAMS (0)
LIN XP283 C_DIS

;ENDFOLD
;FOLD LIN P284 CONT Vel=0.134 m/s CPDATP284 Tool[2] Base[7] ;%{PE}
;FOLD Parameters ;%{h}
;Params IlfProvider=kukaroboter.basistech.inlineforms.movement.old; Kuka.IsGlobalPoint=False; Kuka.PointName=P284; Kuka.BlendingEnabled=TRUE; Kuka.MoveDataName=CPDATP284; Kuka.VelocityPath=0.134; Kuka.CurrentCDSetIndex=0; Kuka.MovementParameterFieldEnabled=True; IlfCommand=LIN
;ENDFOLD
$BWDSTART = FALSE
LDAT_ACT=LCPDATP284
FDAT_ACT=FP284
BAS (#CP_PARAMS,0.134)
SET_CD_PARAMS (0)
LIN XP284 C_DIS

;ENDFOLD
;FOLD LIN P285 CONT Vel=0.134 m/s CPDATP285 Tool[2] Base[7] ;%{PE}
;FOLD Parameters ;%{h}
;Params IlfProvider=kukaroboter.basistech.inlineforms.movement.old; Kuka.IsGlobalPoint=False; Kuka.PointName=P285; Kuka.BlendingEnabled=TRUE; Kuka.MoveDataName=CPDATP285; Kuka.VelocityPath=0.134; Kuka.CurrentCDSetIndex=0; Kuka.MovementParameterFieldEnabled=True; IlfCommand=LIN
;ENDFOLD
$BWDSTART = FALSE
LDAT_ACT=LCPDATP285
FDAT_ACT=FP285
BAS (#CP_PARAMS,0.134)
SET_CD_PARAMS (0)
LIN XP285 C_DIS

;ENDFOLD
;FOLD LIN P286 CONT Vel=0.141 m/s CPDATP286 Tool[2] Base[7] ;%{PE}
;FOLD Parameters ;%{h}
;Params IlfProvider=kukaroboter.basistech.inlineforms.movement.old; Kuka.IsGlobalPoint=False; Kuka.PointName=P286; Kuka.BlendingEnabled=TRUE; Kuka.MoveDataName=CPDATP286; Kuka.VelocityPath=0.141; Kuka.CurrentCDSetIndex=0; Kuka.MovementParameterFieldEnabled=True; IlfCommand=LIN
;ENDFOLD
$BWDSTART = FALSE
LDAT_ACT=LCPDATP286
FDAT_ACT=FP286
BAS (#CP_PARAMS,0.141)
SET_CD_PARAMS (0)
LIN XP286 C_DIS

;ENDFOLD
;FOLD LIN P287 CONT Vel=0.141 m/s CPDATP287 Tool[2] Base[7] ;%{PE}
;FOLD Parameters ;%{h}
;Params IlfProvider=kukaroboter.basistech.inlineforms.movement.old; Kuka.IsGlobalPoint=False; Kuka.PointName=P287; Kuka.BlendingEnabled=TRUE; Kuka.MoveDataName=CPDATP287; Kuka.VelocityPath=0.141; Kuka.CurrentCDSetIndex=0; Kuka.MovementParameterFieldEnabled=True; IlfCommand=LIN
;ENDFOLD
$BWDSTART = FALSE
LDAT_ACT=LCPDATP287
FDAT_ACT=FP287
BAS (#CP_PARAMS,0.141)
SET_CD_PARAMS (0)
LIN XP287 C_DIS

;ENDFOLD
;FOLD LIN P288 CONT Vel=0.141 m/s CPDATP288 Tool[2] Base[7] ;%{PE}
;FOLD Parameters ;%{h}
;Params IlfProvider=kukaroboter.basistech.inlineforms.movement.old; Kuka.IsGlobalPoint=False; Kuka.PointName=P288; Kuka.BlendingEnabled=TRUE; Kuka.MoveDataName=CPDATP288; Kuka.VelocityPath=0.141; Kuka.CurrentCDSetIndex=0; Kuka.MovementParameterFieldEnabled=True; IlfCommand=LIN
;ENDFOLD
$BWDSTART = FALSE
LDAT_ACT=LCPDATP288
FDAT_ACT=FP288
BAS (#CP_PARAMS,0.141)
SET_CD_PARAMS (0)
LIN XP288 C_DIS

;ENDFOLD
;FOLD LIN P289 CONT Vel=0.141 m/s CPDATP289 Tool[2] Base[7] ;%{PE}
;FOLD Parameters ;%{h}
;Params IlfProvider=kukaroboter.basistech.inlineforms.movement.old; Kuka.IsGlobalPoint=False; Kuka.PointName=P289; Kuka.BlendingEnabled=TRUE; Kuka.MoveDataName=CPDATP289; Kuka.VelocityPath=0.141; Kuka.CurrentCDSetIndex=0; Kuka.MovementParameterFieldEnabled=True; IlfCommand=LIN
;ENDFOLD
$BWDSTART = FALSE
LDAT_ACT=LCPDATP289
FDAT_ACT=FP289
BAS (#CP_PARAMS,0.141)
SET_CD_PARAMS (0)
LIN XP289 C_DIS

;ENDFOLD
;FOLD LIN P290 CONT Vel=0.058 m/s CPDATP290 Tool[2] Base[7] ;%{PE}
;FOLD Parameters ;%{h}
;Params IlfProvider=kukaroboter.basistech.inlineforms.movement.old; Kuka.IsGlobalPoint=False; Kuka.PointName=P290; Kuka.BlendingEnabled=TRUE; Kuka.MoveDataName=CPDATP290; Kuka.VelocityPath=0.058; Kuka.CurrentCDSetIndex=0; Kuka.MovementParameterFieldEnabled=True; IlfCommand=LIN
;ENDFOLD
$BWDSTART = FALSE
LDAT_ACT=LCPDATP290
FDAT_ACT=FP290
BAS (#CP_PARAMS,0.058)
SET_CD_PARAMS (0)
LIN XP290 C_DIS

;ENDFOLD
;FOLD LIN P291 CONT Vel=0.058 m/s CPDATP291 Tool[2] Base[7] ;%{PE}
;FOLD Parameters ;%{h}
;Params IlfProvider=kukaroboter.basistech.inlineforms.movement.old; Kuka.IsGlobalPoint=False; Kuka.PointName=P291; Kuka.BlendingEnabled=TRUE; Kuka.MoveDataName=CPDATP291; Kuka.VelocityPath=0.058; Kuka.CurrentCDSetIndex=0; Kuka.MovementParameterFieldEnabled=True; IlfCommand=LIN
;ENDFOLD
$BWDSTART = FALSE
LDAT_ACT=LCPDATP291
FDAT_ACT=FP291
BAS (#CP_PARAMS,0.058)
SET_CD_PARAMS (0)
LIN XP291 C_DIS

;ENDFOLD
;FOLD LIN P292 CONT Vel=0.058 m/s CPDATP292 Tool[2] Base[7] ;%{PE}
;FOLD Parameters ;%{h}
;Params IlfProvider=kukaroboter.basistech.inlineforms.movement.old; Kuka.IsGlobalPoint=False; Kuka.PointName=P292; Kuka.BlendingEnabled=TRUE; Kuka.MoveDataName=CPDATP292; Kuka.VelocityPath=0.058; Kuka.CurrentCDSetIndex=0; Kuka.MovementParameterFieldEnabled=True; IlfCommand=LIN
;ENDFOLD
$BWDSTART = FALSE
LDAT_ACT=LCPDATP292
FDAT_ACT=FP292
BAS (#CP_PARAMS,0.058)
SET_CD_PARAMS (0)
LIN XP292 C_DIS

;ENDFOLD
;FOLD LIN P293 CONT Vel=0.058 m/s CPDATP293 Tool[2] Base[7] ;%{PE}
;FOLD Parameters ;%{h}
;Params IlfProvider=kukaroboter.basistech.inlineforms.movement.old; Kuka.IsGlobalPoint=False; Kuka.PointName=P293; Kuka.BlendingEnabled=TRUE; Kuka.MoveDataName=CPDATP293; Kuka.VelocityPath=0.058; Kuka.CurrentCDSetIndex=0; Kuka.MovementParameterFieldEnabled=True; IlfCommand=LIN
;ENDFOLD
$BWDSTART = FALSE
LDAT_ACT=LCPDATP293
FDAT_ACT=FP293
BAS (#CP_PARAMS,0.058)
SET_CD_PARAMS (0)
LIN XP293 C_DIS

;ENDFOLD
;FOLD LIN P294 CONT Vel=0.127 m/s CPDATP294 Tool[2] Base[7] ;%{PE}
;FOLD Parameters ;%{h}
;Params IlfProvider=kukaroboter.basistech.inlineforms.movement.old; Kuka.IsGlobalPoint=False; Kuka.PointName=P294; Kuka.BlendingEnabled=TRUE; Kuka.MoveDataName=CPDATP294; Kuka.VelocityPath=0.127; Kuka.CurrentCDSetIndex=0; Kuka.MovementParameterFieldEnabled=True; IlfCommand=LIN
;ENDFOLD
$BWDSTART = FALSE
LDAT_ACT=LCPDATP294
FDAT_ACT=FP294
BAS (#CP_PARAMS,0.127)
SET_CD_PARAMS (0)
LIN XP294 C_DIS

;ENDFOLD
;FOLD LIN P295 CONT Vel=0.127 m/s CPDATP295 Tool[2] Base[7] ;%{PE}
;FOLD Parameters ;%{h}
;Params IlfProvider=kukaroboter.basistech.inlineforms.movement.old; Kuka.IsGlobalPoint=False; Kuka.PointName=P295; Kuka.BlendingEnabled=TRUE; Kuka.MoveDataName=CPDATP295; Kuka.VelocityPath=0.127; Kuka.CurrentCDSetIndex=0; Kuka.MovementParameterFieldEnabled=True; IlfCommand=LIN
;ENDFOLD
$BWDSTART = FALSE
LDAT_ACT=LCPDATP295
FDAT_ACT=FP295
BAS (#CP_PARAMS,0.127)
SET_CD_PARAMS (0)
LIN XP295 C_DIS

;ENDFOLD
;FOLD LIN P296 CONT Vel=0.127 m/s CPDATP296 Tool[2] Base[7] ;%{PE}
;FOLD Parameters ;%{h}
;Params IlfProvider=kukaroboter.basistech.inlineforms.movement.old; Kuka.IsGlobalPoint=False; Kuka.PointName=P296; Kuka.BlendingEnabled=TRUE; Kuka.MoveDataName=CPDATP296; Kuka.VelocityPath=0.127; Kuka.CurrentCDSetIndex=0; Kuka.MovementParameterFieldEnabled=True; IlfCommand=LIN
;ENDFOLD
$BWDSTART = FALSE
LDAT_ACT=LCPDATP296
FDAT_ACT=FP296
BAS (#CP_PARAMS,0.127)
SET_CD_PARAMS (0)
LIN XP296 C_DIS

;ENDFOLD
;FOLD LIN P297 CONT Vel=0.127 m/s CPDATP297 Tool[2] Base[7] ;%{PE}
;FOLD Parameters ;%{h}
;Params IlfProvider=kukaroboter.basistech.inlineforms.movement.old; Kuka.IsGlobalPoint=False; Kuka.PointName=P297; Kuka.BlendingEnabled=TRUE; Kuka.MoveDataName=CPDATP297; Kuka.VelocityPath=0.127; Kuka.CurrentCDSetIndex=0; Kuka.MovementParameterFieldEnabled=True; IlfCommand=LIN
;ENDFOLD
$BWDSTART = FALSE
LDAT_ACT=LCPDATP297
FDAT_ACT=FP297
BAS (#CP_PARAMS,0.127)
SET_CD_PARAMS (0)
LIN XP297 C_DIS

;ENDFOLD
;FOLD LIN P298 CONT Vel=0.052 m/s CPDATP298 Tool[2] Base[7] ;%{PE}
;FOLD Parameters ;%{h}
;Params IlfProvider=kukaroboter.basistech.inlineforms.movement.old; Kuka.IsGlobalPoint=False; Kuka.PointName=P298; Kuka.BlendingEnabled=TRUE; Kuka.MoveDataName=CPDATP298; Kuka.VelocityPath=0.052; Kuka.CurrentCDSetIndex=0; Kuka.MovementParameterFieldEnabled=True; IlfCommand=LIN
;ENDFOLD
$BWDSTART = FALSE
LDAT_ACT=LCPDATP298
FDAT_ACT=FP298
BAS (#CP_PARAMS,0.052)
SET_CD_PARAMS (0)
LIN XP298 C_DIS

;ENDFOLD
;FOLD LIN P299 CONT Vel=0.052 m/s CPDATP299 Tool[2] Base[7] ;%{PE}
;FOLD Parameters ;%{h}
;Params IlfProvider=kukaroboter.basistech.inlineforms.movement.old; Kuka.IsGlobalPoint=False; Kuka.PointName=P299; Kuka.BlendingEnabled=TRUE; Kuka.MoveDataName=CPDATP299; Kuka.VelocityPath=0.052; Kuka.CurrentCDSetIndex=0; Kuka.MovementParameterFieldEnabled=True; IlfCommand=LIN
;ENDFOLD
$BWDSTART = FALSE
LDAT_ACT=LCPDATP299
FDAT_ACT=FP299
BAS (#CP_PARAMS,0.052)
SET_CD_PARAMS (0)
LIN XP299 C_DIS

;ENDFOLD
;FOLD LIN P300 CONT Vel=0.052 m/s CPDATP300 Tool[2] Base[7] ;%{PE}
;FOLD Parameters ;%{h}
;Params IlfProvider=kukaroboter.basistech.inlineforms.movement.old; Kuka.IsGlobalPoint=False; Kuka.PointName=P300; Kuka.BlendingEnabled=TRUE; Kuka.MoveDataName=CPDATP300; Kuka.VelocityPath=0.052; Kuka.CurrentCDSetIndex=0; Kuka.MovementParameterFieldEnabled=True; IlfCommand=LIN
;ENDFOLD
$BWDSTART = FALSE
LDAT_ACT=LCPDATP300
FDAT_ACT=FP300
BAS (#CP_PARAMS,0.052)
SET_CD_PARAMS (0)
LIN XP300 C_DIS

;ENDFOLD
;FOLD LIN P301 CONT Vel=0.052 m/s CPDATP301 Tool[2] Base[7] ;%{PE}
;FOLD Parameters ;%{h}
;Params IlfProvider=kukaroboter.basistech.inlineforms.movement.old; Kuka.IsGlobalPoint=False; Kuka.PointName=P301; Kuka.BlendingEnabled=TRUE; Kuka.MoveDataName=CPDATP301; Kuka.VelocityPath=0.052; Kuka.CurrentCDSetIndex=0; Kuka.MovementParameterFieldEnabled=True; IlfCommand=LIN
;ENDFOLD
$BWDSTART = FALSE
LDAT_ACT=LCPDATP301
FDAT_ACT=FP301
BAS (#CP_PARAMS,0.052)
SET_CD_PARAMS (0)
LIN XP301 C_DIS

;ENDFOLD
;FOLD LIN P302 CONT Vel=0.067 m/s CPDATP302 Tool[2] Base[7] ;%{PE}
;FOLD Parameters ;%{h}
;Params IlfProvider=kukaroboter.basistech.inlineforms.movement.old; Kuka.IsGlobalPoint=False; Kuka.PointName=P302; Kuka.BlendingEnabled=TRUE; Kuka.MoveDataName=CPDATP302; Kuka.VelocityPath=0.067; Kuka.CurrentCDSetIndex=0; Kuka.MovementParameterFieldEnabled=True; IlfCommand=LIN
;ENDFOLD
$BWDSTART = FALSE
LDAT_ACT=LCPDATP302
FDAT_ACT=FP302
BAS (#CP_PARAMS,0.067)
SET_CD_PARAMS (0)
LIN XP302 C_DIS

;ENDFOLD
;FOLD LIN P303 CONT Vel=0.067 m/s CPDATP303 Tool[2] Base[7] ;%{PE}
;FOLD Parameters ;%{h}
;Params IlfProvider=kukaroboter.basistech.inlineforms.movement.old; Kuka.IsGlobalPoint=False; Kuka.PointName=P303; Kuka.BlendingEnabled=TRUE; Kuka.MoveDataName=CPDATP303; Kuka.VelocityPath=0.067; Kuka.CurrentCDSetIndex=0; Kuka.MovementParameterFieldEnabled=True; IlfCommand=LIN
;ENDFOLD
$BWDSTART = FALSE
LDAT_ACT=LCPDATP303
FDAT_ACT=FP303
BAS (#CP_PARAMS,0.067)
SET_CD_PARAMS (0)
LIN XP303 C_DIS

;ENDFOLD
;FOLD LIN P304 CONT Vel=0.067 m/s CPDATP304 Tool[2] Base[7] ;%{PE}
;FOLD Parameters ;%{h}
;Params IlfProvider=kukaroboter.basistech.inlineforms.movement.old; Kuka.IsGlobalPoint=False; Kuka.PointName=P304; Kuka.BlendingEnabled=TRUE; Kuka.MoveDataName=CPDATP304; Kuka.VelocityPath=0.067; Kuka.CurrentCDSetIndex=0; Kuka.MovementParameterFieldEnabled=True; IlfCommand=LIN
;ENDFOLD
$BWDSTART = FALSE
LDAT_ACT=LCPDATP304
FDAT_ACT=FP304
BAS (#CP_PARAMS,0.067)
SET_CD_PARAMS (0)
LIN XP304 C_DIS

;ENDFOLD
;FOLD LIN P305 CONT Vel=0.067 m/s CPDATP305 Tool[2] Base[7] ;%{PE}
;FOLD Parameters ;%{h}
;Params IlfProvider=kukaroboter.basistech.inlineforms.movement.old; Kuka.IsGlobalPoint=False; Kuka.PointName=P305; Kuka.BlendingEnabled=TRUE; Kuka.MoveDataName=CPDATP305; Kuka.VelocityPath=0.067; Kuka.CurrentCDSetIndex=0; Kuka.MovementParameterFieldEnabled=True; IlfCommand=LIN
;ENDFOLD
$BWDSTART = FALSE
LDAT_ACT=LCPDATP305
FDAT_ACT=FP305
BAS (#CP_PARAMS,0.067)
SET_CD_PARAMS (0)
LIN XP305 C_DIS

;ENDFOLD
;FOLD LIN P306 CONT Vel=0.117 m/s CPDATP306 Tool[2] Base[7] ;%{PE}
;FOLD Parameters ;%{h}
;Params IlfProvider=kukaroboter.basistech.inlineforms.movement.old; Kuka.IsGlobalPoint=False; Kuka.PointName=P306; Kuka.BlendingEnabled=TRUE; Kuka.MoveDataName=CPDATP306; Kuka.VelocityPath=0.117; Kuka.CurrentCDSetIndex=0; Kuka.MovementParameterFieldEnabled=True; IlfCommand=LIN
;ENDFOLD
$BWDSTART = FALSE
LDAT_ACT=LCPDATP306
FDAT_ACT=FP306
BAS (#CP_PARAMS,0.117)
SET_CD_PARAMS (0)
LIN XP306 C_DIS

;ENDFOLD
;FOLD LIN P307 CONT Vel=0.117 m/s CPDATP307 Tool[2] Base[7] ;%{PE}
;FOLD Parameters ;%{h}
;Params IlfProvider=kukaroboter.basistech.inlineforms.movement.old; Kuka.IsGlobalPoint=False; Kuka.PointName=P307; Kuka.BlendingEnabled=TRUE; Kuka.MoveDataName=CPDATP307; Kuka.VelocityPath=0.117; Kuka.CurrentCDSetIndex=0; Kuka.MovementParameterFieldEnabled=True; IlfCommand=LIN
;ENDFOLD
$BWDSTART = FALSE
LDAT_ACT=LCPDATP307
FDAT_ACT=FP307
BAS (#CP_PARAMS,0.117)
SET_CD_PARAMS (0)
LIN XP307 C_DIS

;ENDFOLD
;FOLD LIN P308 CONT Vel=0.117 m/s CPDATP308 Tool[2] Base[7] ;%{PE}
;FOLD Parameters ;%{h}
;Params IlfProvider=kukaroboter.basistech.inlineforms.movement.old; Kuka.IsGlobalPoint=False; Kuka.PointName=P308; Kuka.BlendingEnabled=TRUE; Kuka.MoveDataName=CPDATP308; Kuka.VelocityPath=0.117; Kuka.CurrentCDSetIndex=0; Kuka.MovementParameterFieldEnabled=True; IlfCommand=LIN
;ENDFOLD
$BWDSTART = FALSE
LDAT_ACT=LCPDATP308
FDAT_ACT=FP308
BAS (#CP_PARAMS,0.117)
SET_CD_PARAMS (0)
LIN XP308 C_DIS

;ENDFOLD
;FOLD LIN P309 CONT Vel=0.117 m/s CPDATP309 Tool[2] Base[7] ;%{PE}
;FOLD Parameters ;%{h}
;Params IlfProvider=kukaroboter.basistech.inlineforms.movement.old; Kuka.IsGlobalPoint=False; Kuka.PointName=P309; Kuka.BlendingEnabled=TRUE; Kuka.MoveDataName=CPDATP309; Kuka.VelocityPath=0.117; Kuka.CurrentCDSetIndex=0; Kuka.MovementParameterFieldEnabled=True; IlfCommand=LIN
;ENDFOLD
$BWDSTART = FALSE
LDAT_ACT=LCPDATP309
FDAT_ACT=FP309
BAS (#CP_PARAMS,0.117)
SET_CD_PARAMS (0)
LIN XP309 C_DIS

;ENDFOLD
;FOLD LIN P310 CONT Vel=0.138 m/s CPDATP310 Tool[2] Base[7] ;%{PE}
;FOLD Parameters ;%{h}
;Params IlfProvider=kukaroboter.basistech.inlineforms.movement.old; Kuka.IsGlobalPoint=False; Kuka.PointName=P310; Kuka.BlendingEnabled=TRUE; Kuka.MoveDataName=CPDATP310; Kuka.VelocityPath=0.138; Kuka.CurrentCDSetIndex=0; Kuka.MovementParameterFieldEnabled=True; IlfCommand=LIN
;ENDFOLD
$BWDSTART = FALSE
LDAT_ACT=LCPDATP310
FDAT_ACT=FP310
BAS (#CP_PARAMS,0.138)
SET_CD_PARAMS (0)
LIN XP310 C_DIS

;ENDFOLD
;FOLD LIN P311 CONT Vel=0.138 m/s CPDATP311 Tool[2] Base[7] ;%{PE}
;FOLD Parameters ;%{h}
;Params IlfProvider=kukaroboter.basistech.inlineforms.movement.old; Kuka.IsGlobalPoint=False; Kuka.PointName=P311; Kuka.BlendingEnabled=TRUE; Kuka.MoveDataName=CPDATP311; Kuka.VelocityPath=0.138; Kuka.CurrentCDSetIndex=0; Kuka.MovementParameterFieldEnabled=True; IlfCommand=LIN
;ENDFOLD
$BWDSTART = FALSE
LDAT_ACT=LCPDATP311
FDAT_ACT=FP311
BAS (#CP_PARAMS,0.138)
SET_CD_PARAMS (0)
LIN XP311 C_DIS

;ENDFOLD
;FOLD LIN P312 CONT Vel=0.138 m/s CPDATP312 Tool[2] Base[7] ;%{PE}
;FOLD Parameters ;%{h}
;Params IlfProvider=kukaroboter.basistech.inlineforms.movement.old; Kuka.IsGlobalPoint=False; Kuka.PointName=P312; Kuka.BlendingEnabled=TRUE; Kuka.MoveDataName=CPDATP312; Kuka.VelocityPath=0.138; Kuka.CurrentCDSetIndex=0; Kuka.MovementParameterFieldEnabled=True; IlfCommand=LIN
;ENDFOLD
$BWDSTART = FALSE
LDAT_ACT=LCPDATP312
FDAT_ACT=FP312
BAS (#CP_PARAMS,0.138)
SET_CD_PARAMS (0)
LIN XP312 C_DIS

;ENDFOLD
;FOLD LIN P313 CONT Vel=0.138 m/s CPDATP313 Tool[2] Base[7] ;%{PE}
;FOLD Parameters ;%{h}
;Params IlfProvider=kukaroboter.basistech.inlineforms.movement.old; Kuka.IsGlobalPoint=False; Kuka.PointName=P313; Kuka.BlendingEnabled=TRUE; Kuka.MoveDataName=CPDATP313; Kuka.VelocityPath=0.138; Kuka.CurrentCDSetIndex=0; Kuka.MovementParameterFieldEnabled=True; IlfCommand=LIN
;ENDFOLD
$BWDSTART = FALSE
LDAT_ACT=LCPDATP313
FDAT_ACT=FP313
BAS (#CP_PARAMS,0.138)
SET_CD_PARAMS (0)
LIN XP313 C_DIS

;ENDFOLD
;FOLD LIN P314 CONT Vel=0.119 m/s CPDATP314 Tool[2] Base[7] ;%{PE}
;FOLD Parameters ;%{h}
;Params IlfProvider=kukaroboter.basistech.inlineforms.movement.old; Kuka.IsGlobalPoint=False; Kuka.PointName=P314; Kuka.BlendingEnabled=TRUE; Kuka.MoveDataName=CPDATP314; Kuka.VelocityPath=0.119; Kuka.CurrentCDSetIndex=0; Kuka.MovementParameterFieldEnabled=True; IlfCommand=LIN
;ENDFOLD
$BWDSTART = FALSE
LDAT_ACT=LCPDATP314
FDAT_ACT=FP314
BAS (#CP_PARAMS,0.119)
SET_CD_PARAMS (0)
LIN XP314 C_DIS

;ENDFOLD
;FOLD LIN P315 CONT Vel=0.119 m/s CPDATP315 Tool[2] Base[7] ;%{PE}
;FOLD Parameters ;%{h}
;Params IlfProvider=kukaroboter.basistech.inlineforms.movement.old; Kuka.IsGlobalPoint=False; Kuka.PointName=P315; Kuka.BlendingEnabled=TRUE; Kuka.MoveDataName=CPDATP315; Kuka.VelocityPath=0.119; Kuka.CurrentCDSetIndex=0; Kuka.MovementParameterFieldEnabled=True; IlfCommand=LIN
;ENDFOLD
$BWDSTART = FALSE
LDAT_ACT=LCPDATP315
FDAT_ACT=FP315
BAS (#CP_PARAMS,0.119)
SET_CD_PARAMS (0)
LIN XP315 C_DIS

;ENDFOLD
;FOLD LIN P316 CONT Vel=0.119 m/s CPDATP316 Tool[2] Base[7] ;%{PE}
;FOLD Parameters ;%{h}
;Params IlfProvider=kukaroboter.basistech.inlineforms.movement.old; Kuka.IsGlobalPoint=False; Kuka.PointName=P316; Kuka.BlendingEnabled=TRUE; Kuka.MoveDataName=CPDATP316; Kuka.VelocityPath=0.119; Kuka.CurrentCDSetIndex=0; Kuka.MovementParameterFieldEnabled=True; IlfCommand=LIN
;ENDFOLD
$BWDSTART = FALSE
LDAT_ACT=LCPDATP316
FDAT_ACT=FP316
BAS (#CP_PARAMS,0.119)
SET_CD_PARAMS (0)
LIN XP316 C_DIS

;ENDFOLD
;FOLD LIN P317 CONT Vel=0.119 m/s CPDATP317 Tool[2] Base[7] ;%{PE}
;FOLD Parameters ;%{h}
;Params IlfProvider=kukaroboter.basistech.inlineforms.movement.old; Kuka.IsGlobalPoint=False; Kuka.PointName=P317; Kuka.BlendingEnabled=TRUE; Kuka.MoveDataName=CPDATP317; Kuka.VelocityPath=0.119; Kuka.CurrentCDSetIndex=0; Kuka.MovementParameterFieldEnabled=True; IlfCommand=LIN
;ENDFOLD
$BWDSTART = FALSE
LDAT_ACT=LCPDATP317
FDAT_ACT=FP317
BAS (#CP_PARAMS,0.119)
SET_CD_PARAMS (0)
LIN XP317 C_DIS

;ENDFOLD
;FOLD LIN P318 CONT Vel=0.121 m/s CPDATP318 Tool[2] Base[7] ;%{PE}
;FOLD Parameters ;%{h}
;Params IlfProvider=kukaroboter.basistech.inlineforms.movement.old; Kuka.IsGlobalPoint=False; Kuka.PointName=P318; Kuka.BlendingEnabled=TRUE; Kuka.MoveDataName=CPDATP318; Kuka.VelocityPath=0.121; Kuka.CurrentCDSetIndex=0; Kuka.MovementParameterFieldEnabled=True; IlfCommand=LIN
;ENDFOLD
$BWDSTART = FALSE
LDAT_ACT=LCPDATP318
FDAT_ACT=FP318
BAS (#CP_PARAMS,0.121)
SET_CD_PARAMS (0)
LIN XP318 C_DIS

;ENDFOLD
;FOLD LIN P319 CONT Vel=0.121 m/s CPDATP319 Tool[2] Base[7] ;%{PE}
;FOLD Parameters ;%{h}
;Params IlfProvider=kukaroboter.basistech.inlineforms.movement.old; Kuka.IsGlobalPoint=False; Kuka.PointName=P319; Kuka.BlendingEnabled=TRUE; Kuka.MoveDataName=CPDATP319; Kuka.VelocityPath=0.121; Kuka.CurrentCDSetIndex=0; Kuka.MovementParameterFieldEnabled=True; IlfCommand=LIN
;ENDFOLD
$BWDSTART = FALSE
LDAT_ACT=LCPDATP319
FDAT_ACT=FP319
BAS (#CP_PARAMS,0.121)
SET_CD_PARAMS (0)
LIN XP319 C_DIS

;ENDFOLD
;FOLD LIN P320 CONT Vel=0.121 m/s CPDATP320 Tool[2] Base[7] ;%{PE}
;FOLD Parameters ;%{h}
;Params IlfProvider=kukaroboter.basistech.inlineforms.movement.old; Kuka.IsGlobalPoint=False; Kuka.PointName=P320; Kuka.BlendingEnabled=TRUE; Kuka.MoveDataName=CPDATP320; Kuka.VelocityPath=0.121; Kuka.CurrentCDSetIndex=0; Kuka.MovementParameterFieldEnabled=True; IlfCommand=LIN
;ENDFOLD
$BWDSTART = FALSE
LDAT_ACT=LCPDATP320
FDAT_ACT=FP320
BAS (#CP_PARAMS,0.121)
SET_CD_PARAMS (0)
LIN XP320 C_DIS

;ENDFOLD
;FOLD LIN P321 CONT Vel=0.121 m/s CPDATP321 Tool[2] Base[7] ;%{PE}
;FOLD Parameters ;%{h}
;Params IlfProvider=kukaroboter.basistech.inlineforms.movement.old; Kuka.IsGlobalPoint=False; Kuka.PointName=P321; Kuka.BlendingEnabled=TRUE; Kuka.MoveDataName=CPDATP321; Kuka.VelocityPath=0.121; Kuka.CurrentCDSetIndex=0; Kuka.MovementParameterFieldEnabled=True; IlfCommand=LIN
;ENDFOLD
$BWDSTART = FALSE
LDAT_ACT=LCPDATP321
FDAT_ACT=FP321
BAS (#CP_PARAMS,0.121)
SET_CD_PARAMS (0)
LIN XP321 C_DIS

;ENDFOLD
;FOLD LIN P322 CONT Vel=0.059 m/s CPDATP322 Tool[2] Base[7] ;%{PE}
;FOLD Parameters ;%{h}
;Params IlfProvider=kukaroboter.basistech.inlineforms.movement.old; Kuka.IsGlobalPoint=False; Kuka.PointName=P322; Kuka.BlendingEnabled=TRUE; Kuka.MoveDataName=CPDATP322; Kuka.VelocityPath=0.059; Kuka.CurrentCDSetIndex=0; Kuka.MovementParameterFieldEnabled=True; IlfCommand=LIN
;ENDFOLD
$BWDSTART = FALSE
LDAT_ACT=LCPDATP322
FDAT_ACT=FP322
BAS (#CP_PARAMS,0.059)
SET_CD_PARAMS (0)
LIN XP322 C_DIS

;ENDFOLD
;FOLD LIN P323 CONT Vel=0.059 m/s CPDATP323 Tool[2] Base[7] ;%{PE}
;FOLD Parameters ;%{h}
;Params IlfProvider=kukaroboter.basistech.inlineforms.movement.old; Kuka.IsGlobalPoint=False; Kuka.PointName=P323; Kuka.BlendingEnabled=TRUE; Kuka.MoveDataName=CPDATP323; Kuka.VelocityPath=0.059; Kuka.CurrentCDSetIndex=0; Kuka.MovementParameterFieldEnabled=True; IlfCommand=LIN
;ENDFOLD
$BWDSTART = FALSE
LDAT_ACT=LCPDATP323
FDAT_ACT=FP323
BAS (#CP_PARAMS,0.059)
SET_CD_PARAMS (0)
LIN XP323 C_DIS

;ENDFOLD
;FOLD LIN P324 CONT Vel=0.059 m/s CPDATP324 Tool[2] Base[7] ;%{PE}
;FOLD Parameters ;%{h}
;Params IlfProvider=kukaroboter.basistech.inlineforms.movement.old; Kuka.IsGlobalPoint=False; Kuka.PointName=P324; Kuka.BlendingEnabled=TRUE; Kuka.MoveDataName=CPDATP324; Kuka.VelocityPath=0.059; Kuka.CurrentCDSetIndex=0; Kuka.MovementParameterFieldEnabled=True; IlfCommand=LIN
;ENDFOLD
$BWDSTART = FALSE
LDAT_ACT=LCPDATP324
FDAT_ACT=FP324
BAS (#CP_PARAMS,0.059)
SET_CD_PARAMS (0)
LIN XP324 C_DIS

;ENDFOLD
;FOLD LIN P325 CONT Vel=0.059 m/s CPDATP325 Tool[2] Base[7] ;%{PE}
;FOLD Parameters ;%{h}
;Params IlfProvider=kukaroboter.basistech.inlineforms.movement.old; Kuka.IsGlobalPoint=False; Kuka.PointName=P325; Kuka.BlendingEnabled=TRUE; Kuka.MoveDataName=CPDATP325; Kuka.VelocityPath=0.059; Kuka.CurrentCDSetIndex=0; Kuka.MovementParameterFieldEnabled=True; IlfCommand=LIN
;ENDFOLD
$BWDSTART = FALSE
LDAT_ACT=LCPDATP325
FDAT_ACT=FP325
BAS (#CP_PARAMS,0.059)
SET_CD_PARAMS (0)
LIN XP325 C_DIS

;ENDFOLD
;FOLD LIN P326 CONT Vel=0.08 m/s CPDATP326 Tool[2] Base[7] ;%{PE}
;FOLD Parameters ;%{h}
;Params IlfProvider=kukaroboter.basistech.inlineforms.movement.old; Kuka.IsGlobalPoint=False; Kuka.PointName=P326; Kuka.BlendingEnabled=TRUE; Kuka.MoveDataName=CPDATP326; Kuka.VelocityPath=0.08; Kuka.CurrentCDSetIndex=0; Kuka.MovementParameterFieldEnabled=True; IlfCommand=LIN
;ENDFOLD
$BWDSTART = FALSE
LDAT_ACT=LCPDATP326
FDAT_ACT=FP326
BAS (#CP_PARAMS,0.08)
SET_CD_PARAMS (0)
LIN XP326 C_DIS

;ENDFOLD
;FOLD LIN P327 CONT Vel=0.08 m/s CPDATP327 Tool[2] Base[7] ;%{PE}
;FOLD Parameters ;%{h}
;Params IlfProvider=kukaroboter.basistech.inlineforms.movement.old; Kuka.IsGlobalPoint=False; Kuka.PointName=P327; Kuka.BlendingEnabled=TRUE; Kuka.MoveDataName=CPDATP327; Kuka.VelocityPath=0.08; Kuka.CurrentCDSetIndex=0; Kuka.MovementParameterFieldEnabled=True; IlfCommand=LIN
;ENDFOLD
$BWDSTART = FALSE
LDAT_ACT=LCPDATP327
FDAT_ACT=FP327
BAS (#CP_PARAMS,0.08)
SET_CD_PARAMS (0)
LIN XP327 C_DIS

;ENDFOLD
;FOLD LIN P328 CONT Vel=0.08 m/s CPDATP328 Tool[2] Base[7] ;%{PE}
;FOLD Parameters ;%{h}
;Params IlfProvider=kukaroboter.basistech.inlineforms.movement.old; Kuka.IsGlobalPoint=False; Kuka.PointName=P328; Kuka.BlendingEnabled=TRUE; Kuka.MoveDataName=CPDATP328; Kuka.VelocityPath=0.08; Kuka.CurrentCDSetIndex=0; Kuka.MovementParameterFieldEnabled=True; IlfCommand=LIN
;ENDFOLD
$BWDSTART = FALSE
LDAT_ACT=LCPDATP328
FDAT_ACT=FP328
BAS (#CP_PARAMS,0.08)
SET_CD_PARAMS (0)
LIN XP328 C_DIS

;ENDFOLD
;FOLD LIN P329 CONT Vel=0.08 m/s CPDATP329 Tool[2] Base[7] ;%{PE}
;FOLD Parameters ;%{h}
;Params IlfProvider=kukaroboter.basistech.inlineforms.movement.old; Kuka.IsGlobalPoint=False; Kuka.PointName=P329; Kuka.BlendingEnabled=TRUE; Kuka.MoveDataName=CPDATP329; Kuka.VelocityPath=0.08; Kuka.CurrentCDSetIndex=0; Kuka.MovementParameterFieldEnabled=True; IlfCommand=LIN
;ENDFOLD
$BWDSTART = FALSE
LDAT_ACT=LCPDATP329
FDAT_ACT=FP329
BAS (#CP_PARAMS,0.08)
SET_CD_PARAMS (0)
LIN XP329 C_DIS

;ENDFOLD
;FOLD LIN P330 CONT Vel=0.136 m/s CPDATP330 Tool[2] Base[7] ;%{PE}
;FOLD Parameters ;%{h}
;Params IlfProvider=kukaroboter.basistech.inlineforms.movement.old; Kuka.IsGlobalPoint=False; Kuka.PointName=P330; Kuka.BlendingEnabled=TRUE; Kuka.MoveDataName=CPDATP330; Kuka.VelocityPath=0.136; Kuka.CurrentCDSetIndex=0; Kuka.MovementParameterFieldEnabled=True; IlfCommand=LIN
;ENDFOLD
$BWDSTART = FALSE
LDAT_ACT=LCPDATP330
FDAT_ACT=FP330
BAS (#CP_PARAMS,0.136)
SET_CD_PARAMS (0)
LIN XP330 C_DIS

;ENDFOLD
;FOLD LIN P331 CONT Vel=0.136 m/s CPDATP331 Tool[2] Base[7] ;%{PE}
;FOLD Parameters ;%{h}
;Params IlfProvider=kukaroboter.basistech.inlineforms.movement.old; Kuka.IsGlobalPoint=False; Kuka.PointName=P331; Kuka.BlendingEnabled=TRUE; Kuka.MoveDataName=CPDATP331; Kuka.VelocityPath=0.136; Kuka.CurrentCDSetIndex=0; Kuka.MovementParameterFieldEnabled=True; IlfCommand=LIN
;ENDFOLD
$BWDSTART = FALSE
LDAT_ACT=LCPDATP331
FDAT_ACT=FP331
BAS (#CP_PARAMS,0.136)
SET_CD_PARAMS (0)
LIN XP331 C_DIS

;ENDFOLD
;FOLD LIN P332 CONT Vel=0.136 m/s CPDATP332 Tool[2] Base[7] ;%{PE}
;FOLD Parameters ;%{h}
;Params IlfProvider=kukaroboter.basistech.inlineforms.movement.old; Kuka.IsGlobalPoint=False; Kuka.PointName=P332; Kuka.BlendingEnabled=TRUE; Kuka.MoveDataName=CPDATP332; Kuka.VelocityPath=0.136; Kuka.CurrentCDSetIndex=0; Kuka.MovementParameterFieldEnabled=True; IlfCommand=LIN
;ENDFOLD
$BWDSTART = FALSE
LDAT_ACT=LCPDATP332
FDAT_ACT=FP332
BAS (#CP_PARAMS,0.136)
SET_CD_PARAMS (0)
LIN XP332 C_DIS

;ENDFOLD
;FOLD LIN P333 CONT Vel=0.136 m/s CPDATP333 Tool[2] Base[7] ;%{PE}
;FOLD Parameters ;%{h}
;Params IlfProvider=kukaroboter.basistech.inlineforms.movement.old; Kuka.IsGlobalPoint=False; Kuka.PointName=P333; Kuka.BlendingEnabled=TRUE; Kuka.MoveDataName=CPDATP333; Kuka.VelocityPath=0.136; Kuka.CurrentCDSetIndex=0; Kuka.MovementParameterFieldEnabled=True; IlfCommand=LIN
;ENDFOLD
$BWDSTART = FALSE
LDAT_ACT=LCPDATP333
FDAT_ACT=FP333
BAS (#CP_PARAMS,0.136)
SET_CD_PARAMS (0)
LIN XP333 C_DIS

;ENDFOLD
;FOLD LIN P334 CONT Vel=0.5 m/s CPDATP334 Tool[2] Base[7] ;%{PE}
;FOLD Parameters ;%{h}
;Params IlfProvider=kukaroboter.basistech.inlineforms.movement.old; Kuka.IsGlobalPoint=False; Kuka.PointName=P334; Kuka.BlendingEnabled=TRUE; Kuka.MoveDataName=CPDATP334; Kuka.VelocityPath=0.5; Kuka.CurrentCDSetIndex=0; Kuka.MovementParameterFieldEnabled=True; IlfCommand=LIN
;ENDFOLD
$BWDSTART = FALSE
LDAT_ACT=LCPDATP334
FDAT_ACT=FP334
BAS (#CP_PARAMS,0.5)
SET_CD_PARAMS (0)
LIN XP334 C_DIS

;ENDFOLD
;FOLD LIN P335 CONT Vel=1.0 m/s CPDATP335 Tool[2] Base[7] ;%{PE}
;FOLD Parameters ;%{h}
;Params IlfProvider=kukaroboter.basistech.inlineforms.movement.old; Kuka.IsGlobalPoint=False; Kuka.PointName=P335; Kuka.BlendingEnabled=TRUE; Kuka.MoveDataName=CPDATP335; Kuka.VelocityPath=1.0; Kuka.CurrentCDSetIndex=0; Kuka.MovementParameterFieldEnabled=True; IlfCommand=LIN
;ENDFOLD
$BWDSTART = FALSE
LDAT_ACT=LCPDATP335
FDAT_ACT=FP335
BAS (#CP_PARAMS,1.0)
SET_CD_PARAMS (0)
LIN XP335 C_DIS

;ENDFOLD
;FOLD LIN P336 CONT Vel=1.0 m/s CPDATP336 Tool[2] Base[7] ;%{PE}
;FOLD Parameters ;%{h}
;Params IlfProvider=kukaroboter.basistech.inlineforms.movement.old; Kuka.IsGlobalPoint=False; Kuka.PointName=P336; Kuka.BlendingEnabled=TRUE; Kuka.MoveDataName=CPDATP336; Kuka.VelocityPath=1.0; Kuka.CurrentCDSetIndex=0; Kuka.MovementParameterFieldEnabled=True; IlfCommand=LIN
;ENDFOLD
$BWDSTART = FALSE
LDAT_ACT=LCPDATP336
FDAT_ACT=FP336
BAS (#CP_PARAMS,1.0)
SET_CD_PARAMS (0)
LIN XP336 C_DIS

;ENDFOLD
END
;End of routine {i}

--- Inconel_dataset.dat ---
&ACCESS RVP1
&REL 1217
&PARAM WOPTRAJECTORYID = 2
&PARAM WOPTEMPLATENAME = WopCoreTemplatePath
&PARAM DISKPATH = KRC:\R1\Program\Working Paths
DEFDAT  Inconel_dataset
;FOLD EXTERNAL DECLARATIONS;%{PE}%MKUKATPBASIS,%CEXT,%VCOMMON,%P
;FOLD BASISTECH EXT;%{PE}%MKUKATPBASIS,%CEXT,%VEXT,%P
EXT  BAS (BAS_COMMAND  :IN,REAL  :IN )
DECL INT SUCCESS
;ENDFOLD (BASISTECH EXT)
;FOLD USER EXT;%{E}%MKUKATPUSER,%CEXT,%VEXT,%P
;Make your modifications here

;ENDFOLD (USER EXT)
;ENDFOLD (EXTERNAL DECLARATIONS)

INT APP_GENNUMBER = 215375
INT APP_ANSWER
INT APP_OFFSET
DECL STATE_T APP_STATE

DECL PDAT PPDATP0={VEL 100,ACC 100,APO_DIST 5,APO_MODE #CDIS,GEAR_JERK 100.0,EXAX_IGN 0}
DECL FDAT FP0={TOOL_NO 2,BASE_NO 10,IPO_FRAME #BASE,POINT2[] " ",TQ_STATE FALSE}
DECL E6AXIS XP0={A1 -1000.000,A2 -90.000,A3 90.000,A4 0.000,A5 -90.000,A6 0.000,E1 0.000,E2 -41.000,E3 33.000,E4 0.000,E5 0.000,E6 0.000}

; Data for Routine_0
DECL LDAT LCPDATP1={VEL 1.0,ACC 100,APO_DIST 5,APO_FAC 50.0,ORI_TYP #VAR,CIRC_TYP #BASE,JERK_FAC 50.0}
DECL FDAT FP1={TOOL_NO 2,BASE_NO 10,IPO_FRAME #BASE,POINT2[] " ",TQ_STATE FALSE}
DECL E6POS XP1={X 100.000,Y 0.000,Z -100.000,A 0.000,B 0.000,C 0.000}
DECL LDAT LCPDATP2={VEL 0.116,ACC 100,APO_DIST 5,APO_FAC 50.0,ORI_TYP #VAR,CIRC_TYP #BASE,JERK_FAC 50.0}
DECL FDAT FP2={TOOL_NO 2,BASE_NO 10,IPO_FRAME #BASE,POINT2[] " ",TQ_STATE FALSE}
DECL E6POS XP2={X 50.000,Y -5.730,Z -30.020,A 0.000,B 0.000,C -28.000}
DECL LDAT LCPDATP3={VEL 0.116,ACC 100,APO_DIST 5,APO_FAC 50.0,ORI_TYP #VAR,CIRC_TYP #BASE,JERK_FAC 50.0}
DECL FDAT FP3={TOOL_NO 2,BASE_NO 10,IPO_FRAME #BASE,POINT2[] " ",TQ_STATE FALSE}
DECL E6POS XP3={X 0.000,Y -5.730,Z -30.020,A 0.000,B 0.000,C -28.000}
DECL LDAT LCPDATP4={VEL 0.116,ACC 100,APO_DIST 5,APO_FAC 50.0,ORI_TYP #VAR,CIRC_TYP #BASE,JERK_FAC 50.0}
DECL FDAT FP4={TOOL_NO 2,BASE_NO 10,IPO_FRAME #BASE,POINT2[] " ",TQ_STATE FALSE}
DECL E6POS XP4={X -50.000,Y -5.730,Z -30.020,A 0.000,B 0.000,C -28.000}
DECL LDAT LCPDATP5={VEL 0.116,ACC 100,APO_DIST 5,APO_FAC 50.0,ORI_TYP #VAR,CIRC_TYP #BASE,JERK_FAC 50.0}
DECL FDAT FP5={TOOL_NO 2,BASE_NO 10,IPO_FRAME #BASE,POINT2[] " ",TQ_STATE FALSE}
DECL E6POS XP5={X -100.000,Y -5.730,Z -30.020,A 0.000,B 0.000,C -28.000}
DECL LDAT LCPDATP6={VEL 0.099,ACC 100,APO_DIST 5,APO_FAC 50.0,ORI_TYP #VAR,CIRC_TYP #BASE,JERK_FAC 50.0}
DECL FDAT FP6={TOOL_NO 2,BASE_NO 10,IPO_FRAME #BASE,POINT2[] " ",TQ_STATE FALSE}
DECL E6POS XP6={X -100.000,Y 4.550,Z -24.510,A 0.000,B 0.000,C -40.000}
DECL LDAT LCPDATP7={VEL 0.099,ACC 100,APO_DIST 5,APO_FAC 50.0,ORI_TYP #VAR,CIRC_TYP #BASE,JERK_FAC 50.0}
DECL FDAT FP7={TOOL_NO 2,BASE_NO 10,IPO_FRAME #BASE,POINT2[] " ",TQ_STATE FALSE}
DECL E6POS XP7={X -50.000,Y 4.550,Z -24.510,A 0.000,B 0.000,C -40.000}
DECL LDAT LCPDATP8={VEL 0.099,ACC 100,APO_DIST 5,APO_FAC 50.0,ORI_TYP #VAR,CIRC_TYP #BASE,JERK_FAC 50.0}
DECL FDAT FP8={TOOL_NO 2,BASE_NO 10,IPO_FRAME #BASE,POINT2[] " ",TQ_STATE FALSE}
DECL E6POS XP8={X -0.000,Y 4.550,Z -24.510,A 0.000,B 0.000,C -40.000}
DECL LDAT LCPDATP9={VEL 0.099,ACC 100,APO_DIST 5,APO_FAC 50.0,ORI_TYP #VAR,CIRC_TYP #BASE,JERK_FAC 50.0}
DECL FDAT FP9={TOOL_NO 2,BASE_NO 10,IPO_FRAME #BASE,POINT2[] " ",TQ_STATE FALSE}
DECL E6POS XP9={X 50.000,Y 4.550,Z -24.510,A 0.000,B 0.000,C -40.000}
DECL LDAT LCPDATP10={VEL 0.075,ACC 100,APO_DIST 5,APO_FAC 50.0,ORI_TYP #VAR,CIRC_TYP #BASE,JERK_FAC 50.0}
DECL FDAT FP10={TOOL_NO 2,BASE_NO 10,IPO_FRAME #BASE,POINT2[] " ",TQ_STATE FALSE}
DECL E6POS XP10={X 50.000,Y 24.940,Z -36.820,A 0.000,B 0.000,C -23.000}
DECL LDAT LCPDATP11={VEL 0.075,ACC 100,APO_DIST 5,APO_FAC 50.0,ORI_TYP #VAR,CIRC_TYP #BASE,JERK_FAC 50.0}
DECL FDAT FP11={TOOL_NO 2,BASE_NO 10,IPO_FRAME #BASE,POINT2[] " ",TQ_STATE FALSE}
DECL E6POS XP11={X -0.000,Y 24.940,Z -36.820,A 0.000,B 0.000,C -23.000}
DECL LDAT LCPDATP12={VEL 0.075,ACC 100,APO_DIST 5,APO_FAC 50.0,ORI_TYP #VAR,CIRC_TYP #BASE,JERK_FAC 50.0}
DECL FDAT FP12={TOOL_NO 2,BASE_NO 10,IPO_FRAME #BASE,POINT2[] " ",TQ_STATE FALSE}
DECL E6POS XP12={X -50.000,Y 24.940,Z -36.820,A 0.000,B 0.000,C -23.000}
DECL LDAT LCPDATP13={VEL 0.075,ACC 100,APO_DIST 5,APO_FAC 50.0,ORI_TYP #VAR,CIRC_TYP #BASE,JERK_FAC 50.0}
DECL FDAT FP13={TOOL_NO 2,BASE_NO 10,IPO_FRAME #BASE,POINT2[] " ",TQ_STATE FALSE}
DECL E6POS XP13={X -100.000,Y 24.940,Z -36.820,A 0.000,B 0.000,C -23.000}
DECL LDAT LCPDATP14={VEL 0.113,ACC 100,APO_DIST 5,APO_FAC 50.0,ORI_TYP #VAR,CIRC_TYP #BASE,JERK_FAC 50.0}
DECL FDAT FP14={TOOL_NO 2,BASE_NO 10,IPO_FRAME #BASE,POINT2[] " ",TQ_STATE FALSE}
DECL E6POS XP14={X -100.000,Y 52.180,Z -87.790,A 0.000,B 0.000,C -4.000}
DECL LDAT LCPDATP15={VEL 0.113,ACC 100,APO_DIST 5,APO_FAC 50.0,ORI_TYP #VAR,CIRC_TYP #BASE,JERK_FAC 50.0}
DECL FDAT FP15={TOOL_NO 2,BASE_NO 10,IPO_FRAME #BASE,POINT2[] " ",TQ_STATE FALSE}
DECL E6POS XP15={X -50.000,Y 52.180,Z -87.790,A 0.000,B 0.000,C -4.000}
DECL LDAT LCPDATP16={VEL 0.113,ACC 100,APO_DIST 5,APO_FAC 50.0,ORI_TYP #VAR,CIRC_TYP #BASE,JERK_FAC 50.0}
DECL FDAT FP16={TOOL_NO 2,BASE_NO 10,IPO_FRAME #BASE,POINT2[] " ",TQ_STATE FALSE}
DECL E6POS XP16={X -0.000,Y 52.180,Z -87.790,A 0.000,B 0.000,C -4.000}
DECL LDAT LCPDATP17={VEL 0.113,ACC 100,APO_DIST 5,APO_FAC 50.0,ORI_TYP #VAR,CIRC_TYP #BASE,JERK_FAC 50.0}
DECL FDAT FP17={TOOL_NO 2,BASE_NO 10,IPO_FRAME #BASE,POINT2[] " ",TQ_STATE FALSE}
DECL E6POS XP17={X 50.000,Y 52.180,Z -87.790,A 0.000,B 0.000,C -4.000}
DECL LDAT LCPDATP18={VEL 0.086,ACC 100,APO_DIST 5,APO_FAC 50.0,ORI_TYP #VAR,CIRC_TYP #BASE,JERK_FAC 50.0}
DECL FDAT FP18={TOOL_NO 2,BASE_NO 10,IPO_FRAME #BASE,POINT2[] " ",TQ_STATE FALSE}
DECL E6POS XP18={X 50.000,Y 68.620,Z -69.900,A 0.000,B 0.000,C -3.000}
DECL LDAT LCPDATP19={VEL 0.086,ACC 100,APO_DIST 5,APO_FAC 50.0,ORI_TYP #VAR,CIRC_TYP #BASE,JERK_FAC 50.0}
DECL FDAT FP19={TOOL_NO 2,BASE_NO 10,IPO_FRAME #BASE,POINT2[] " ",TQ_STATE FALSE}
DECL E6POS XP19={X -0.000,Y 68.620,Z -69.900,A 0.000,B 0.000,C -3.000}
DECL LDAT LCPDATP20={VEL 0.086,ACC 100,APO_DIST 5,APO_FAC 50.0,ORI_TYP #VAR,CIRC_TYP #BASE,JERK_FAC 50.0}
DECL FDAT FP20={TOOL_NO 2,BASE_NO 10,IPO_FRAME #BASE,POINT2[] " ",TQ_STATE FALSE}
DECL E6POS XP20={X -50.000,Y 68.620,Z -69.900,A 0.000,B 0.000,C -3.000}
DECL LDAT LCPDATP21={VEL 0.086,ACC 100,APO_DIST 5,APO_FAC 50.0,ORI_TYP #VAR,CIRC_TYP #BASE,JERK_FAC 50.0}
DECL FDAT FP21={TOOL_NO 2,BASE_NO 10,IPO_FRAME #BASE,POINT2[] " ",TQ_STATE FALSE}
DECL E6POS XP21={X -100.000,Y 68.620,Z -69.900,A 0.000,B 0.000,C -3.000}
DECL LDAT LCPDATP22={VEL 0.073,ACC 100,APO_DIST 5,APO_FAC 50.0,ORI_TYP #VAR,CIRC_TYP #BASE,JERK_FAC 50.0}
DECL FDAT FP22={TOOL_NO 2,BASE_NO 10,IPO_FRAME #BASE,POINT2[] " ",TQ_STATE FALSE}
DECL E6POS XP22={X -100.000,Y 65.180,Z -95.090,A 0.000,B 0.000,C -14.000}
DECL LDAT LCPDATP23={VEL 0.073,ACC 100,APO_DIST 5,APO_FAC 50.0,ORI_TYP #VAR,CIRC_TYP #BASE,JERK_FAC 50.0}
DECL FDAT FP23={TOOL_NO 2,BASE_NO 10,IPO_FRAME #BASE,POINT2[] " ",TQ_STATE FALSE}
DECL E6POS XP23={X -50.000,Y 65.180,Z -95.090,A 0.000,B 0.000,C -14.000}
DECL LDAT LCPDATP24={VEL 0.073,ACC 100,APO_DIST 5,APO_FAC 50.0,ORI_TYP #VAR,CIRC_TYP #BASE,JERK_FAC 50.0}
DECL FDAT FP24={TOOL_NO 2,BASE_NO 10,IPO_FRAME #BASE,POINT2[] " ",TQ_STATE FALSE}
DECL E6POS XP24={X -0.000,Y 65.180,Z -95.090,A 0.000,B 0.000,C -14.000}
DECL LDAT LCPDATP25={VEL 0.073,ACC 100,APO_DIST 5,APO_FAC 50.0,ORI_TYP #VAR,CIRC_TYP #BASE,JERK_FAC 50.0}
DECL FDAT FP25={TOOL_NO 2,BASE_NO 10,IPO_FRAME #BASE,POINT2[] " ",TQ_STATE FALSE}
DECL E6POS XP25={X 50.000,Y 65.180,Z -95.090,A 0.000,B 0.000,C -14.000}
DECL LDAT LCPDATP26={VEL 0.137,ACC 100,APO_DIST 5,APO_FAC 50.0,ORI_TYP #VAR,CIRC_TYP #BASE,JERK_FAC 50.0}
DECL FDAT FP26={TOOL_NO 2,BASE_NO 10,IPO_FRAME #BASE,POINT2[] " ",TQ_STATE FALSE}
DECL E6POS XP26={X 50.000,Y 48.190,Z -79.460,A 0.000,B 0.000,C -35.000}
DECL LDAT LCPDATP27={VEL 0.137,ACC 100,APO_DIST 5,APO_FAC 50.0,ORI_TYP #VAR,CIRC_TYP #BASE,JERK_FAC 50.0}
DECL FDAT FP27={TOOL_NO 2,BASE_NO 10,IPO_FRAME #BASE,POINT2[] " ",TQ_STATE FALSE}
DECL E6POS XP27={X -0.000,Y 48.190,Z -79.460,A 0.000,B 0.000,C -35.000}
DECL LDAT LCPDATP28={VEL 0.137,ACC 100,APO_DIST 5,APO_FAC 50.0,ORI_TYP #VAR,CIRC_TYP #BASE,JERK_FAC 50.0}
DECL FDAT FP28={TOOL_NO 2,BASE_NO 10,IPO_FRAME #BASE,POINT2[] " ",TQ_STATE FALSE}
DECL E6POS XP28={X -50.000,Y 48.190,Z -79.460,A 0.000,B 0.000,C -35.000}
DECL LDAT LCPDATP29={VEL 0.137,ACC 100,APO_DIST 5,APO_FAC 50.0,ORI_TYP #VAR,CIRC_TYP #BASE,JERK_FAC 50.0}
DECL FDAT FP29={TOOL_NO 2,BASE_NO 10,IPO_FRAME #BASE,POINT2[] " ",TQ_STATE FALSE}
DECL E6POS XP29={X -100.000,Y 48.190,Z -79.460,A 0.000,B 0.000,C -35.000}
DECL LDAT LCPDATP30={VEL 0.082,ACC 100,APO_DIST 5,APO_FAC 50.0,ORI_TYP #VAR,CIRC_TYP #BASE,JERK_FAC 50.0}
DECL FDAT FP30={TOOL_NO 2,BASE_NO 10,IPO_FRAME #BASE,POINT2[] " ",TQ_STATE FALSE}
DECL E6POS XP30={X -100.000,Y 87.280,Z -46.640,A 0.000,B 0.000,C -32.000}
DECL LDAT LCPDATP31={VEL 0.082,ACC 100,APO_DIST 5,APO_FAC 50.0,ORI_TYP #VAR,CIRC_TYP #BASE,JERK_FAC 50.0}
DECL FDAT FP31={TOOL_NO 2,BASE_NO 10,IPO_FRAME #BASE,POINT2[] " ",TQ_STATE FALSE}
DECL E6POS XP31={X -50.000,Y 87.280,Z -46.640,A 0.000,B 0.000,C -32.000}
DECL LDAT LCPDATP32={VEL 0.082,ACC 100,APO_DIST 5,APO_FAC 50.0,ORI_TYP #VAR,CIRC_TYP #BASE,JERK_FAC 50.0}
DECL FDAT FP32={TOOL_NO 2,BASE_NO 10,IPO_FRAME #BASE,POINT2[] " ",TQ_STATE FALSE}
DECL E6POS XP32={X -0.000,Y 87.280,Z -46.640,A 0.000,B 0.000,C -32.000}
DECL LDAT LCPDATP33={VEL 0.082,ACC 100,APO_DIST 5,APO_FAC 50.0,ORI_TYP #VAR,CIRC_TYP #BASE,JERK_FAC 50.0}
DECL FDAT FP33={TOOL_NO 2,BASE_NO 10,IPO_FRAME #BASE,POINT2[] " ",TQ_STATE FALSE}
DECL E6POS XP33={X 50.000,Y 87.280,Z -46.640,A 0.000,B 0.000,C -32.000}
DECL LDAT LCPDATP34={VEL 0.086,ACC 100,APO_DIST 5,APO_FAC 50.0,ORI_TYP #VAR,CIRC_TYP #BASE,JERK_FAC 50.0}
DECL FDAT FP34={TOOL_NO 2,BASE_NO 10,IPO_FRAME #BASE,POINT2[] " ",TQ_STATE FALSE}
DECL E6POS XP34={X 50.000,Y 101.710,Z -93.610,A 0.000,B 0.000,C -19.000}
DECL LDAT LCPDATP35={VEL 0.086,ACC 100,APO_DIST 5,APO_FAC 50.0,ORI_TYP #VAR,CIRC_TYP #BASE,JERK_FAC 50.0}
DECL FDAT FP35={TOOL_NO 2,BASE_NO 10,IPO_FRAME #BASE,POINT2[] " ",TQ_STATE FALSE}
DECL E6POS XP35={X -0.000,Y 101.710,Z -93.610,A 0.000,B 0.000,C -19.000}
DECL LDAT LCPDATP36={VEL 0.086,ACC 100,APO_DIST 5,APO_FAC 50.0,ORI_TYP #VAR,CIRC_TYP #BASE,JERK_FAC 50.0}
DECL FDAT FP36={TOOL_NO 2,BASE_NO 10,IPO_FRAME #BASE,POINT2[] " ",TQ_STATE FALSE}
DECL E6POS XP36={X -50.000,Y 101.710,Z -93.610,A 0.000,B 0.000,C -19.000}
DECL LDAT LCPDATP37={VEL 0.086,ACC 100,APO_DIST 5,APO_FAC 50.0,ORI_TYP #VAR,CIRC_TYP #BASE,JERK_FAC 50.0}
DECL FDAT FP37={TOOL_NO 2,BASE_NO 10,IPO_FRAME #BASE,POINT2[] " ",TQ_STATE FALSE}
DECL E6POS XP37={X -100.000,Y 101.710,Z -93.610,A 0.000,B 0.000,C -19.000}
DECL LDAT LCPDATP38={VEL 0.097,ACC 100,APO_DIST 5,APO_FAC 50.0,ORI_TYP #VAR,CIRC_TYP #BASE,JERK_FAC 50.0}
DECL FDAT FP38={TOOL_NO 2,BASE_NO 10,IPO_FRAME #BASE,POINT2[] " ",TQ_STATE FALSE}
DECL E6POS XP38={X -100.000,Y 117.680,Z -79.350,A 0.000,B 0.000,C -21.000}
DECL LDAT LCPDATP39={VEL 0.097,ACC 100,APO_DIST 5,APO_FAC 50.0,ORI_TYP #VAR,CIRC_TYP #BASE,JERK_FAC 50.0}
DECL FDAT FP39={TOOL_NO 2,BASE_NO 10,IPO_FRAME #BASE,POINT2[] " ",TQ_STATE FALSE}
DECL E6POS XP39={X -50.000,Y 117.680,Z -79.350,A 0.000,B 0.000,C -21.000}
DECL LDAT LCPDATP40={VEL 0.097,ACC 100,APO_DIST 5,APO_FAC 50.0,ORI_TYP #VAR,CIRC_TYP #BASE,JERK_FAC 50.0}
DECL FDAT FP40={TOOL_NO 2,BASE_NO 10,IPO_FRAME #BASE,POINT2[] " ",TQ_STATE FALSE}
DECL E6POS XP40={X -0.000,Y 117.680,Z -79.350,A 0.000,B 0.000,C -21.000}
DECL LDAT LCPDATP41={VEL 0.097,ACC 100,APO_DIST 5,APO_FAC 50.0,ORI_TYP #VAR,CIRC_TYP #BASE,JERK_FAC 50.0}
DECL FDAT FP41={TOOL_NO 2,BASE_NO 10,IPO_FRAME #BASE,POINT2[] " ",TQ_STATE FALSE}
DECL E6POS XP41={X 50.000,Y 117.680,Z -79.350,A 0.000,B 0.000,C -21.000}
DECL LDAT LCPDATP42={VEL 0.136,ACC 100,APO_DIST 5,APO_FAC 50.0,ORI_TYP #VAR,CIRC_TYP #BASE,JERK_FAC 50.0}
DECL FDAT FP42={TOOL_NO 2,BASE_NO 10,IPO_FRAME #BASE,POINT2[] " ",TQ_STATE FALSE}
DECL E6POS XP42={X 50.000,Y 150.480,Z -65.980,A 0.000,B 0.000,C -10.000}
DECL LDAT LCPDATP43={VEL 0.136,ACC 100,APO_DIST 5,APO_FAC 50.0,ORI_TYP #VAR,CIRC_TYP #BASE,JERK_FAC 50.0}
DECL FDAT FP43={TOOL_NO 2,BASE_NO 10,IPO_FRAME #BASE,POINT2[] " ",TQ_STATE FALSE}
DECL E6POS XP43={X -0.000,Y 150.480,Z -65.980,A 0.000,B 0.000,C -10.000}
DECL LDAT LCPDATP44={VEL 0.136,ACC 100,APO_DIST 5,APO_FAC 50.0,ORI_TYP #VAR,CIRC_TYP #BASE,JERK_FAC 50.0}
DECL FDAT FP44={TOOL_NO 2,BASE_NO 10,IPO_FRAME #BASE,POINT2[] " ",TQ_STATE FALSE}
DECL E6POS XP44={X -50.000,Y 150.480,Z -65.980,A 0.000,B 0.000,C -10.000}
DECL LDAT LCPDATP45={VEL 0.136,ACC 100,APO_DIST 5,APO_FAC 50.0,ORI_TYP #VAR,CIRC_TYP #BASE,JERK_FAC 50.0}
DECL FDAT FP45={TOOL_NO 2,BASE_NO 10,IPO_FRAME #BASE,POINT2[] " ",TQ_STATE FALSE}
DECL E6POS XP45={X -100.000,Y 150.480,Z -65.980,A 0.000,B 0.000,C -10.000}
DECL LDAT LCPDATP46={VEL 0.107,ACC 100,APO_DIST 5,APO_FAC 50.0,ORI_TYP #VAR,CIRC_TYP #BASE,JERK_FAC 50.0}
DECL FDAT FP46={TOOL_NO 2,BASE_NO 10,IPO_FRAME #BASE,POINT2[] " ",TQ_STATE FALSE}
DECL E6POS XP46={X -100.000,Y 132.510,Z -57.520,A 0.000,B 0.000,C -38.000}
DECL LDAT LCPDATP47={VEL 0.107,ACC 100,APO_DIST 5,APO_FAC 50.0,ORI_TYP #VAR,CIRC_TYP #BASE,JERK_FAC 50.0}
DECL FDAT FP47={TOOL_NO 2,BASE_NO 10,IPO_FRAME #BASE,POINT2[] " ",TQ_STATE FALSE}
DECL E6POS XP47={X -50.000,Y 132.510,Z -57.520,A 0.000,B 0.000,C -38.000}
DECL LDAT LCPDATP48={VEL 0.107,ACC 100,APO_DIST 5,APO_FAC 50.0,ORI_TYP #VAR,CIRC_TYP #BASE,JERK_FAC 50.0}
DECL FDAT FP48={TOOL_NO 2,BASE_NO 10,IPO_FRAME #BASE,POINT2[] " ",TQ_STATE FALSE}
DECL E6POS XP48={X -0.000,Y 132.510,Z -57.520,A 0.000,B 0.000,C -38.000}
DECL LDAT LCPDATP49={VEL 0.107,ACC 100,APO_DIST 5,APO_FAC 50.0,ORI_TYP #VAR,CIRC_TYP #BASE,JERK_FAC 50.0}
DECL FDAT FP49={TOOL_NO 2,BASE_NO 10,IPO_FRAME #BASE,POINT2[] " ",TQ_STATE FALSE}
DECL E6POS XP49={X 50.000,Y 132.510,Z -57.520,A 0.000,B 0.000,C -38.000}
DECL LDAT LCPDATP50={VEL 0.09,ACC 100,APO_DIST 5,APO_FAC 50.0,ORI_TYP #VAR,CIRC_TYP #BASE,JERK_FAC 50.0}
DECL FDAT FP50={TOOL_NO 2,BASE_NO 10,IPO_FRAME #BASE,POINT2[] " ",TQ_STATE FALSE}
DECL E6POS XP50={X 50.000,Y 148.310,Z -68.770,A 0.000,B 0.000,C -33.000}
DECL LDAT LCPDATP51={VEL 0.09,ACC 100,APO_DIST 5,APO_FAC 50.0,ORI_TYP #VAR,CIRC_TYP #BASE,JERK_FAC 50.0}
DECL FDAT FP51={TOOL_NO 2,BASE_NO 10,IPO_FRAME #BASE,POINT2[] " ",TQ_STATE FALSE}
DECL E6POS XP51={X -0.000,Y 148.310,Z -68.770,A 0.000,B 0.000,C -33.000}
DECL LDAT LCPDATP52={VEL 0.09,ACC 100,APO_DIST 5,APO_FAC 50.0,ORI_TYP #VAR,CIRC_TYP #BASE,JERK_FAC 50.0}
DECL FDAT FP52={TOOL_NO 2,BASE_NO 10,IPO_FRAME #BASE,POINT2[] " ",TQ_STATE FALSE}
DECL E6POS XP52={X -50.000,Y 148.310,Z -68.770,A 0.000,B 0.000,C -33.000}
DECL LDAT LCPDATP53={VEL 0.09,ACC 100,APO_DIST 5,APO_FAC 50.0,ORI_TYP #VAR,CIRC_TYP #BASE,JERK_FAC 50.0}
DECL FDAT FP53={TOOL_NO 2,BASE_NO 10,IPO_FRAME #BASE,POINT2[] " ",TQ_STATE FALSE}
DECL E6POS XP53={X -100.000,Y 148.310,Z -68.770,A 0.000,B 0.000,C -33.000}
DECL LDAT LCPDATP54={VEL 0.132,ACC 100,APO_DIST 5,APO_FAC 50.0,ORI_TYP #VAR,CIRC_TYP #BASE,JERK_FAC 50.0}
DECL FDAT FP54={TOOL_NO 2,BASE_NO 10,IPO_FRAME #BASE,POINT2[] " ",TQ_STATE FALSE}
DECL E6POS XP54={X -100.000,Y 203.750,Z -95.870,A 0.000,B 0.000,C -3.000}
DECL LDAT LCPDATP55={VEL 0.132,ACC 100,APO_DIST 5,APO_FAC 50.0,ORI_TYP #VAR,CIRC_TYP #BASE,JERK_FAC 50.0}
DECL FDAT FP55={TOOL_NO 2,BASE_NO 10,IPO_FRAME #BASE,POINT2[] " ",TQ_STATE FALSE}
DECL E6POS XP55={X -50.000,Y 203.750,Z -95.870,A 0.000,B 0.000,C -3.000}
DECL LDAT LCPDATP56={VEL 0.132,ACC 100,APO_DIST 5,APO_FAC 50.0,ORI_TYP #VAR,CIRC_TYP #BASE,JERK_FAC 50.0}
DECL FDAT FP56={TOOL_NO 2,BASE_NO 10,IPO_FRAME #BASE,POINT2[] " ",TQ_STATE FALSE}
DECL E6POS XP56={X -0.000,Y 203.750,Z -95.870,A 0.000,B 0.000,C -3.000}
DECL LDAT LCPDATP57={VEL 0.132,ACC 100,APO_DIST 5,APO_FAC 50.0,ORI_TYP #VAR,CIRC_TYP #BASE,JERK_FAC 50.0}
DECL FDAT FP57={TOOL_NO 2,BASE_NO 10,IPO_FRAME #BASE,POINT2[] " ",TQ_STATE FALSE}
DECL E6POS XP57={X 50.000,Y 203.750,Z -95.870,A 0.000,B 0.000,C -3.000}
DECL LDAT LCPDATP58={VEL 0.068,ACC 100,APO_DIST 5,APO_FAC 50.0,ORI_TYP #VAR,CIRC_TYP #BASE,JERK_FAC 50.0}
DECL FDAT FP58={TOOL_NO 2,BASE_NO 10,IPO_FRAME #BASE,POINT2[] " ",TQ_STATE FALSE}
DECL E6POS XP58={X 50.000,Y 221.500,Z -80.990,A 0.000,B 0.000,C -1.000}
DECL LDAT LCPDATP59={VEL 0.068,ACC 100,APO_DIST 5,APO_FAC 50.0,ORI_TYP #VAR,CIRC_TYP #BASE,JERK_FAC 50.0}
DECL FDAT FP59={TOOL_NO 2,BASE_NO 10,IPO_FRAME #BASE,POINT2[] " ",TQ_STATE FALSE}
DECL E6POS XP59={X -0.000,Y 221.500,Z -80.990,A 0.000,B 0.000,C -1.000}
DECL LDAT LCPDATP60={VEL 0.068,ACC 100,APO_DIST 5,APO_FAC 50.0,ORI_TYP #VAR,CIRC_TYP #BASE,JERK_FAC 50.0}
DECL FDAT FP60={TOOL_NO 2,BASE_NO 10,IPO_FRAME #BASE,POINT2[] " ",TQ_STATE FALSE}
DECL E6POS XP60={X -50.000,Y 221.500,Z -80.990,A 0.000,B 0.000,C -1.000}
DECL LDAT LCPDATP61={VEL 0.068,ACC 100,APO_DIST 5,APO_FAC 50.0,ORI_TYP #VAR,CIRC_TYP #BASE,JERK_FAC 50.0}
DECL FDAT FP61={TOOL_NO 2,BASE_NO 10,IPO_FRAME #BASE,POINT2[] " ",TQ_STATE FALSE}
DECL E6POS XP61={X -100.000,Y 221.500,Z -80.990,A 0.000,B 0.000,C -1.000}
DECL LDAT LCPDATP62={VEL 0.115,ACC 100,APO_DIST 5,APO_FAC 50.0,ORI_TYP #VAR,CIRC_TYP #BASE,JERK_FAC 50.0}
DECL FDAT FP62={TOOL_NO 2,BASE_NO 10,IPO_FRAME #BASE,POINT2[] " ",TQ_STATE FALSE}
DECL E6POS XP62={X -100.000,Y 206.270,Z -52.830,A 0.000,B 0.000,C -30.000}
DECL LDAT LCPDATP63={VEL 0.115,ACC 100,APO_DIST 5,APO_FAC 50.0,ORI_TYP #VAR,CIRC_TYP #BASE,JERK_FAC 50.0}
DECL FDAT FP63={TOOL_NO 2,BASE_NO 10,IPO_FRAME #BASE,POINT2[] " ",TQ_STATE FALSE}
DECL E6POS XP63={X -50.000,Y 206.270,Z -52.830,A 0.000,B 0.000,C -30.000}
DECL LDAT LCPDATP64={VEL 0.115,ACC 100,APO_DIST 5,APO_FAC 50.0,ORI_TYP #VAR,CIRC_TYP #BASE,JERK_FAC 50.0}
DECL FDAT FP64={TOOL_NO 2,BASE_NO 10,IPO_FRAME #BASE,POINT2[] " ",TQ_STATE FALSE}
DECL E6POS XP64={X -0.000,Y 206.270,Z -52.830,A 0.000,B 0.000,C -30.000}
DECL LDAT LCPDATP65={VEL 0.115,ACC 100,APO_DIST 5,APO_FAC 50.0,ORI_TYP #VAR,CIRC_TYP #BASE,JERK_FAC 50.0}
DECL FDAT FP65={TOOL_NO 2,BASE_NO 10,IPO_FRAME #BASE,POINT2[] " ",TQ_STATE FALSE}
DECL E6POS XP65={X 50.000,Y 206.270,Z -52.830,A 0.000,B 0.000,C -30.000}
DECL LDAT LCPDATP66={VEL 0.111,ACC 100,APO_DIST 5,APO_FAC 50.0,ORI_TYP #VAR,CIRC_TYP #BASE,JERK_FAC 50.0}
DECL FDAT FP66={TOOL_NO 2,BASE_NO 10,IPO_FRAME #BASE,POINT2[] " ",TQ_STATE FALSE}
DECL E6POS XP66={X 50.000,Y 214.030,Z -89.530,A 0.000,B 0.000,C -24.000}
DECL LDAT LCPDATP67={VEL 0.111,ACC 100,APO_DIST 5,APO_FAC 50.0,ORI_TYP #VAR,CIRC_TYP #BASE,JERK_FAC 50.0}
DECL FDAT FP67={TOOL_NO 2,BASE_NO 10,IPO_FRAME #BASE,POINT2[] " ",TQ_STATE FALSE}
DECL E6POS XP67={X -0.000,Y 214.030,Z -89.530,A 0.000,B 0.000,C -24.000}
DECL LDAT LCPDATP68={VEL 0.111,ACC 100,APO_DIST 5,APO_FAC 50.0,ORI_TYP #VAR,CIRC_TYP #BASE,JERK_FAC 50.0}
DECL FDAT FP68={TOOL_NO 2,BASE_NO 10,IPO_FRAME #BASE,POINT2[] " ",TQ_STATE FALSE}
DECL E6POS XP68={X -50.000,Y 214.030,Z -89.530,A 0.000,B 0.000,C -24.000}
DECL LDAT LCPDATP69={VEL 0.111,ACC 100,APO_DIST 5,APO_FAC 50.0,ORI_TYP #VAR,CIRC_TYP #BASE,JERK_FAC 50.0}
DECL FDAT FP69={TOOL_NO 2,BASE_NO 10,IPO_FRAME #BASE,POINT2[] " ",TQ_STATE FALSE}
DECL E6POS XP69={X -100.000,Y 214.030,Z -89.530,A 0.000,B 0.000,C -24.000}
DECL LDAT LCPDATP70={VEL 0.124,ACC 100,APO_DIST 5,APO_FAC 50.0,ORI_TYP #VAR,CIRC_TYP #BASE,JERK_FAC 50.0}
DECL FDAT FP70={TOOL_NO 2,BASE_NO 10,IPO_FRAME #BASE,POINT2[] " ",TQ_STATE FALSE}
DECL E6POS XP70={X -100.000,Y 264.220,Z -41.970,A 0.000,B 0.000,C -2.000}
DECL LDAT LCPDATP71={VEL 0.124,ACC 100,APO_DIST 5,APO_FAC 50.0,ORI_TYP #VAR,CIRC_TYP #BASE,JERK_FAC 50.0}
DECL FDAT FP71={TOOL_NO 2,BASE_NO 10,IPO_FRAME #BASE,POINT2[] " ",TQ_STATE FALSE}
DECL E6POS XP71={X -50.000,Y 264.220,Z -41.970,A 0.000,B 0.000,C -2.000}
DECL LDAT LCPDATP72={VEL 0.124,ACC 100,APO_DIST 5,APO_FAC 50.0,ORI_TYP #VAR,CIRC_TYP #BASE,JERK_FAC 50.0}
DECL FDAT FP72={TOOL_NO 2,BASE_NO 10,IPO_FRAME #BASE,POINT2[] " ",TQ_STATE FALSE}
DECL E6POS XP72={X -0.000,Y 264.220,Z -41.970,A 0.000,B 0.000,C -2.000}
DECL LDAT LCPDATP73={VEL 0.124,ACC 100,APO_DIST 5,APO_FAC 50.0,ORI_TYP #VAR,CIRC_TYP #BASE,JERK_FAC 50.0}
DECL FDAT FP73={TOOL_NO 2,BASE_NO 10,IPO_FRAME #BASE,POINT2[] " ",TQ_STATE FALSE}
DECL E6POS XP73={X 50.000,Y 264.220,Z -41.970,A 0.000,B 0.000,C -2.000}
DECL LDAT LCPDATP74={VEL 0.112,ACC 100,APO_DIST 5,APO_FAC 50.0,ORI_TYP #VAR,CIRC_TYP #BASE,JERK_FAC 50.0}
DECL FDAT FP74={TOOL_NO 2,BASE_NO 10,IPO_FRAME #BASE,POINT2[] " ",TQ_STATE FALSE}
DECL E6POS XP74={X 50.000,Y 254.510,Z -62.120,A 0.000,B 0.000,C -24.000}
DECL LDAT LCPDATP75={VEL 0.112,ACC 100,APO_DIST 5,APO_FAC 50.0,ORI_TYP #VAR,CIRC_TYP #BASE,JERK_FAC 50.0}
DECL FDAT FP75={TOOL_NO 2,BASE_NO 10,IPO_FRAME #BASE,POINT2[] " ",TQ_STATE FALSE}
DECL E6POS XP75={X -0.000,Y 254.510,Z -62.120,A 0.000,B 0.000,C -24.000}
DECL LDAT LCPDATP76={VEL 0.112,ACC 100,APO_DIST 5,APO_FAC 50.0,ORI_TYP #VAR,CIRC_TYP #BASE,JERK_FAC 50.0}
DECL FDAT FP76={TOOL_NO 2,BASE_NO 10,IPO_FRAME #BASE,POINT2[] " ",TQ_STATE FALSE}
DECL E6POS XP76={X -50.000,Y 254.510,Z -62.120,A 0.000,B 0.000,C -24.000}
DECL LDAT LCPDATP77={VEL 0.112,ACC 100,APO_DIST 5,APO_FAC 50.0,ORI_TYP #VAR,CIRC_TYP #BASE,JERK_FAC 50.0}
DECL FDAT FP77={TOOL_NO 2,BASE_NO 10,IPO_FRAME #BASE,POINT2[] " ",TQ_STATE FALSE}
DECL E6POS XP77={X -100.000,Y 254.510,Z -62.120,A 0.000,B 0.000,C -24.000}
DECL LDAT LCPDATP78={VEL 0.109,ACC 100,APO_DIST 5,APO_FAC 50.0,ORI_TYP #VAR,CIRC_TYP #BASE,JERK_FAC 50.0}
DECL FDAT FP78={TOOL_NO 2,BASE_NO 10,IPO_FRAME #BASE,POINT2[] " ",TQ_STATE FALSE}
DECL E6POS XP78={X -100.000,Y 269.410,Z -36.410,A 0.000,B 0.000,C -36.000}
DECL LDAT LCPDATP79={VEL 0.109,ACC 100,APO_DIST 5,APO_FAC 50.0,ORI_TYP #VAR,CIRC_TYP #BASE,JERK_FAC 50.0}
DECL FDAT FP79={TOOL_NO 2,BASE_NO 10,IPO_FRAME #BASE,POINT2[] " ",TQ_STATE FALSE}
DECL E6POS XP79={X -50.000,Y 269.410,Z -36.410,A 0.000,B 0.000,C -36.000}
DECL LDAT LCPDATP80={VEL 0.109,ACC 100,APO_DIST 5,APO_FAC 50.0,ORI_TYP #VAR,CIRC_TYP #BASE,JERK_FAC 50.0}
DECL FDAT FP80={TOOL_NO 2,BASE_NO 10,IPO_FRAME #BASE,POINT2[] " ",TQ_STATE FALSE}
DECL E6POS XP80={X -0.000,Y 269.410,Z -36.410,A 0.000,B 0.000,C -36.000}
DECL LDAT LCPDATP81={VEL 0.109,ACC 100,APO_DIST 5,APO_FAC 50.0,ORI_TYP #VAR,CIRC_TYP #BASE,JERK_FAC 50.0}
DECL FDAT FP81={TOOL_NO 2,BASE_NO 10,IPO_FRAME #BASE,POINT2[] " ",TQ_STATE FALSE}
DECL E6POS XP81={X 50.000,Y 269.410,Z -36.410,A 0.000,B 0.000,C -36.000}
DECL LDAT LCPDATP82={VEL 0.104,ACC 100,APO_DIST 5,APO_FAC 50.0,ORI_TYP #VAR,CIRC_TYP #BASE,JERK_FAC 50.0}
DECL FDAT FP82={TOOL_NO 2,BASE_NO 10,IPO_FRAME #BASE,POINT2[] " ",TQ_STATE FALSE}
DECL E6POS XP82={X 50.000,Y 288.080,Z -43.260,A 0.000,B 0.000,C -28.000}
DECL LDAT LCPDATP83={VEL 0.104,ACC 100,APO_DIST 5,APO_FAC 50.0,ORI_TYP #VAR,CIRC_TYP #BASE,JERK_FAC 50.0}
DECL FDAT FP83={TOOL_NO 2,BASE_NO 10,IPO_FRAME #BASE,POINT2[] " ",TQ_STATE FALSE}
DECL E6POS XP83={X -0.000,Y 288.080,Z -43.260,A 0.000,B 0.000,C -28.000}
DECL LDAT LCPDATP84={VEL 0.104,ACC 100,APO_DIST 5,APO_FAC 50.0,ORI_TYP #VAR,CIRC_TYP #BASE,JERK_FAC 50.0}
DECL FDAT FP84={TOOL_NO 2,BASE_NO 10,IPO_FRAME #BASE,POINT2[] " ",TQ_STATE FALSE}
DECL E6POS XP84={X -50.000,Y 288.080,Z -43.260,A 0.000,B 0.000,C -28.000}
DECL LDAT LCPDATP85={VEL 0.104,ACC 100,APO_DIST 5,APO_FAC 50.0,ORI_TYP #VAR,CIRC_TYP #BASE,JERK_FAC 50.0}
DECL FDAT FP85={TOOL_NO 2,BASE_NO 10,IPO_FRAME #BASE,POINT2[] " ",TQ_STATE FALSE}
DECL E6POS XP85={X -100.000,Y 288.080,Z -43.260,A 0.000,B 0.000,C -28.000}
DECL LDAT LCPDATP86={VEL 0.053,ACC 100,APO_DIST 5,APO_FAC 50.0,ORI_TYP #VAR,CIRC_TYP #BASE,JERK_FAC 50.0}
DECL FDAT FP86={TOOL_NO 2,BASE_NO 10,IPO_FRAME #BASE,POINT2[] " ",TQ_STATE FALSE}
DECL E6POS XP86={X -100.000,Y 303.890,Z -73.230,A 0.000,B 0.000,C -18.000}
DECL LDAT LCPDATP87={VEL 0.053,ACC 100,APO_DIST 5,APO_FAC 50.0,ORI_TYP #VAR,CIRC_TYP #BASE,JERK_FAC 50.0}
DECL FDAT FP87={TOOL_NO 2,BASE_NO 10,IPO_FRAME #BASE,POINT2[] " ",TQ_STATE FALSE}
DECL E6POS XP87={X -50.000,Y 303.890,Z -73.230,A 0.000,B 0.000,C -18.000}
DECL LDAT LCPDATP88={VEL 0.053,ACC 100,APO_DIST 5,APO_FAC 50.0,ORI_TYP #VAR,CIRC_TYP #BASE,JERK_FAC 50.0}
DECL FDAT FP88={TOOL_NO 2,BASE_NO 10,IPO_FRAME #BASE,POINT2[] " ",TQ_STATE FALSE}
DECL E6POS XP88={X -0.000,Y 303.890,Z -73.230,A 0.000,B 0.000,C -18.000}
DECL LDAT LCPDATP89={VEL 0.053,ACC 100,APO_DIST 5,APO_FAC 50.0,ORI_TYP #VAR,CIRC_TYP #BASE,JERK_FAC 50.0}
DECL FDAT FP89={TOOL_NO 2,BASE_NO 10,IPO_FRAME #BASE,POINT2[] " ",TQ_STATE FALSE}
DECL E6POS XP89={X 50.000,Y 303.890,Z -73.230,A 0.000,B 0.000,C -18.000}
DECL LDAT LCPDATP90={VEL 0.063,ACC 100,APO_DIST 5,APO_FAC 50.0,ORI_TYP #VAR,CIRC_TYP #BASE,JERK_FAC 50.0}
DECL FDAT FP90={TOOL_NO 2,BASE_NO 10,IPO_FRAME #BASE,POINT2[] " ",TQ_STATE FALSE}
DECL E6POS XP90={X 50.000,Y 335.430,Z -94.640,A 0.000,B 0.000,C -5.000}
DECL LDAT LCPDATP91={VEL 0.063,ACC 100,APO_DIST 5,APO_FAC 50.0,ORI_TYP #VAR,CIRC_TYP #BASE,JERK_FAC 50.0}
DECL FDAT FP91={TOOL_NO 2,BASE_NO 10,IPO_FRAME #BASE,POINT2[] " ",TQ_STATE FALSE}
DECL E6POS XP91={X -0.000,Y 335.430,Z -94.640,A 0.000,B 0.000,C -5.000}
DECL LDAT LCPDATP92={VEL 0.063,ACC 100,APO_DIST 5,APO_FAC 50.0,ORI_TYP #VAR,CIRC_TYP #BASE,JERK_FAC 50.0}
DECL FDAT FP92={TOOL_NO 2,BASE_NO 10,IPO_FRAME #BASE,POINT2[] " ",TQ_STATE FALSE}
DECL E6POS XP92={X -50.000,Y 335.430,Z -94.640,A 0.000,B 0.000,C -5.000}
DECL LDAT LCPDATP93={VEL 0.063,ACC 100,APO_DIST 5,APO_FAC 50.0,ORI_TYP #VAR,CIRC_TYP #BASE,JERK_FAC 50.0}
DECL FDAT FP93={TOOL_NO 2,BASE_NO 10,IPO_FRAME #BASE,POINT2[] " ",TQ_STATE FALSE}
DECL E6POS XP93={X -100.000,Y 335.430,Z -94.640,A 0.000,B 0.000,C -5.000}
DECL LDAT LCPDATP94={VEL 0.5,ACC 100,APO_DIST 5,APO_FAC 50.0,ORI_TYP #VAR,CIRC_TYP #BASE,JERK_FAC 50.0}
DECL FDAT FP94={TOOL_NO 2,BASE_NO 10,IPO_FRAME #BASE,POINT2[] " ",TQ_STATE FALSE}
DECL E6POS XP94={X -150.000,Y 343.710,Z -50.000,A 0.000,B 0.000,C 0.000}
DECL LDAT LCPDATP95={VEL 1.0,ACC 100,APO_DIST 5,APO_FAC 50.0,ORI_TYP #VAR,CIRC_TYP #BASE,JERK_FAC 50.0}
DECL FDAT FP95={TOOL_NO 2,BASE_NO 10,IPO_FRAME #BASE,POINT2[] " ",TQ_STATE FALSE}
DECL E6POS XP95={X -150.000,Y 380.000,Z -20.000,A 0.000,B 0.000,C 0.000}
DECL LDAT LCPDATP96={VEL 1.0,ACC 100,APO_DIST 5,APO_FAC 50.0,ORI_TYP #VAR,CIRC_TYP #BASE,JERK_FAC 50.0}
DECL FDAT FP96={TOOL_NO 2,BASE_NO 10,IPO_FRAME #BASE,POINT2[] " ",TQ_STATE FALSE}
DECL E6POS XP96={X 100.000,Y 380.000,Z -20.000,A 0.000,B 0.000,C 0.000}
;ENDDAT for Routine_0


